(* Logix 5000 project; controller reports 1756-L63 rev 20.15; software revision 20.04; part 12 of 52 *)

        [360].log_data[14].valid := 1, [360].log_data[15].valid := 1, [360].log_data[16].valid := 1, [360].log_data[17].valid := 1, [360].log_data[18].valid := 1, [360].log_data[19].valid := 1, [360].time.Year := 2023, [360].time.Month := 1, [360].time.Day := 19, [360].time.Hour := 6, [360].time.Minute := 24, [360].time.Second := 59, [361].log_data[0].min := 1.0, [361].log_data[0].max := 1.0, [361].log_data[0].total := 300.0, [361].log_data[0].time := 300.0, [361].log_data[0].minminute := 25, [361].log_data[0].maxminute := 25, [361].log_data[0].valid := 1, [361].log_data[1].valid := 1, [361].log_data[2].valid := 1, [361].log_data[3].valid := 1, [361].log_data[4].valid := 1, [361].log_data[5].valid := 1, [361].log_data[6].valid := 1, [361].log_data[7].valid := 1, [361].log_data[8].valid := 1, [361].log_data[9].valid := 1, [361].log_data[10].valid := 1, [361].log_data[11].valid := 1, [361].log_data[12].valid := 1, [361].log_data[13].valid := 1, [361].log_data[14].valid := 1, [361].log_data[15].valid := 1, [361].log_data[16].valid := 1, [361].log_data[17].valid := 1, [361].log_data[18].valid := 1, [361].log_data[19].valid := 1, [361].time.Year := 2023, [361].time.Month := 1, [361].time.Day := 19, [361].time.Hour := 6, [361].time.Minute := 29, [361].time.Second := 59, [362].log_data[0].min := 1.0, [362].log_data[0].max := 1.0, [362].log_data[0].total := 300.0, [362].log_data[0].time := 300.0, [362].log_data[0].minminute := 30, [362].log_data[0].maxminute := 30, [362].log_data[0].valid := 1, [362].log_data[1].valid := 1, [362].log_data[2].valid := 1, [362].log_data[3].valid := 1, [362].log_data[4].valid := 1, [362].log_data[5].valid := 1, [362].log_data[6].valid := 1, [362].log_data[7].valid := 1, [362].log_data[8].valid := 1, [362].log_data[9].valid := 1,
        [362].log_data[10].valid := 1, [362].log_data[11].valid := 1, [362].log_data[12].valid := 1, [362].log_data[13].valid := 1, [362].log_data[14].valid := 1, [362].log_data[15].valid := 1, [362].log_data[16].valid := 1, [362].log_data[17].valid := 1, [362].log_data[18].valid := 1, [362].log_data[19].valid := 1, [362].time.Year := 2023, [362].time.Month := 1, [362].time.Day := 19, [362].time.Hour := 6, [362].time.Minute := 34, [362].time.Second := 59, [363].log_data[0].min := 1.0, [363].log_data[0].max := 1.0, [363].log_data[0].total := 300.0, [363].log_data[0].time := 300.0, [363].log_data[0].minminute := 35, [363].log_data[0].maxminute := 35, [363].log_data[0].valid := 1, [363].log_data[1].valid := 1, [363].log_data[2].valid := 1, [363].log_data[3].valid := 1, [363].log_data[4].valid := 1, [363].log_data[5].valid := 1, [363].log_data[6].valid := 1, [363].log_data[7].valid := 1, [363].log_data[8].valid := 1, [363].log_data[9].valid := 1, [363].log_data[10].valid := 1, [363].log_data[11].valid := 1, [363].log_data[12].valid := 1, [363].log_data[13].valid := 1, [363].log_data[14].valid := 1, [363].log_data[15].valid := 1, [363].log_data[16].valid := 1, [363].log_data[17].valid := 1, [363].log_data[18].valid := 1, [363].log_data[19].valid := 1, [363].time.Year := 2023, [363].time.Month := 1, [363].time.Day := 19, [363].time.Hour := 6, [363].time.Minute := 39, [363].time.Second := 59, [364].log_data[0].min := 1.0, [364].log_data[0].max := 1.0, [364].log_data[0].total := 300.0, [364].log_data[0].time := 300.0, [364].log_data[0].minminute := 40, [364].log_data[0].maxminute := 40, [364].log_data[0].valid := 1, [364].log_data[1].valid := 1, [364].log_data[2].valid := 1, [364].log_data[3].valid := 1, [364].log_data[4].valid := 1, [364].log_data[5].valid := 1,
        [364].log_data[6].valid := 1, [364].log_data[7].valid := 1, [364].log_data[8].valid := 1, [364].log_data[9].valid := 1, [364].log_data[10].valid := 1, [364].log_data[11].valid := 1, [364].log_data[12].valid := 1, [364].log_data[13].valid := 1, [364].log_data[14].valid := 1, [364].log_data[15].valid := 1, [364].log_data[16].valid := 1, [364].log_data[17].valid := 1, [364].log_data[18].valid := 1, [364].log_data[19].valid := 1, [364].time.Year := 2023, [364].time.Month := 1, [364].time.Day := 19, [364].time.Hour := 6, [364].time.Minute := 44, [364].time.Second := 59, [365].log_data[0].min := 1.0, [365].log_data[0].max := 1.0, [365].log_data[0].total := 300.0, [365].log_data[0].time := 300.0, [365].log_data[0].minminute := 45, [365].log_data[0].maxminute := 45, [365].log_data[0].valid := 1, [365].log_data[1].valid := 1, [365].log_data[2].valid := 1, [365].log_data[3].valid := 1, [365].log_data[4].valid := 1, [365].log_data[5].valid := 1, [365].log_data[6].valid := 1, [365].log_data[7].valid := 1, [365].log_data[8].valid := 1, [365].log_data[9].valid := 1, [365].log_data[10].valid := 1, [365].log_data[11].valid := 1, [365].log_data[12].valid := 1, [365].log_data[13].valid := 1, [365].log_data[14].valid := 1, [365].log_data[15].valid := 1, [365].log_data[16].valid := 1, [365].log_data[17].valid := 1, [365].log_data[18].valid := 1, [365].log_data[19].valid := 1, [365].time.Year := 2023, [365].time.Month := 1, [365].time.Day := 19, [365].time.Hour := 6, [365].time.Minute := 49, [365].time.Second := 59, [366].log_data[0].min := 1.0, [366].log_data[0].max := 1.0, [366].log_data[0].total := 300.0, [366].log_data[0].time := 300.0, [366].log_data[0].minminute := 50, [366].log_data[0].maxminute := 50, [366].log_data[0].valid := 1, [366].log_data[1].valid := 1,
        [366].log_data[2].valid := 1, [366].log_data[3].valid := 1, [366].log_data[4].valid := 1, [366].log_data[5].valid := 1, [366].log_data[6].valid := 1, [366].log_data[7].valid := 1, [366].log_data[8].valid := 1, [366].log_data[9].valid := 1, [366].log_data[10].valid := 1, [366].log_data[11].valid := 1, [366].log_data[12].valid := 1, [366].log_data[13].valid := 1, [366].log_data[14].valid := 1, [366].log_data[15].valid := 1, [366].log_data[16].valid := 1, [366].log_data[17].valid := 1, [366].log_data[18].valid := 1, [366].log_data[19].valid := 1, [366].time.Year := 2023, [366].time.Month := 1, [366].time.Day := 19, [366].time.Hour := 6, [366].time.Minute := 54, [366].time.Second := 59, [367].log_data[0].min := 1.0, [367].log_data[0].max := 1.0, [367].log_data[0].total := 300.0, [367].log_data[0].time := 300.0, [367].log_data[0].minminute := 55, [367].log_data[0].maxminute := 55, [367].log_data[0].valid := 1, [367].log_data[1].valid := 1, [367].log_data[2].valid := 1, [367].log_data[3].valid := 1, [367].log_data[4].valid := 1, [367].log_data[5].valid := 1, [367].log_data[6].valid := 1, [367].log_data[7].valid := 1, [367].log_data[8].valid := 1, [367].log_data[9].valid := 1, [367].log_data[10].valid := 1, [367].log_data[11].valid := 1, [367].log_data[12].valid := 1, [367].log_data[13].valid := 1, [367].log_data[14].valid := 1, [367].log_data[15].valid := 1, [367].log_data[16].valid := 1, [367].log_data[17].valid := 1, [367].log_data[18].valid := 1, [367].log_data[19].valid := 1, [367].time.Year := 2023, [367].time.Month := 1, [367].time.Day := 19, [367].time.Hour := 6, [367].time.Minute := 59, [367].time.Second := 59, [368].log_data[0].min := 1.0, [368].log_data[0].max := 1.0, [368].log_data[0].total := 300.0, [368].log_data[0].time := 300.0,
        [368].log_data[0].valid := 1, [368].log_data[1].valid := 1, [368].log_data[2].valid := 1, [368].log_data[3].valid := 1, [368].log_data[4].valid := 1, [368].log_data[5].valid := 1, [368].log_data[6].valid := 1, [368].log_data[7].valid := 1, [368].log_data[8].valid := 1, [368].log_data[9].valid := 1, [368].log_data[10].valid := 1, [368].log_data[11].valid := 1, [368].log_data[12].valid := 1, [368].log_data[13].valid := 1, [368].log_data[14].valid := 1, [368].log_data[15].valid := 1, [368].log_data[16].valid := 1, [368].log_data[17].valid := 1, [368].log_data[18].valid := 1, [368].log_data[19].valid := 1, [368].time.Year := 2023, [368].time.Month := 1, [368].time.Day := 19, [368].time.Hour := 7, [368].time.Minute := 4, [368].time.Second := 59, [369].log_data[0].min := 1.0, [369].log_data[0].max := 1.0, [369].log_data[0].total := 300.0, [369].log_data[0].time := 300.0, [369].log_data[0].minminute := 5, [369].log_data[0].maxminute := 5, [369].log_data[0].valid := 1, [369].log_data[1].valid := 1, [369].log_data[2].valid := 1, [369].log_data[3].valid := 1, [369].log_data[4].valid := 1, [369].log_data[5].valid := 1, [369].log_data[6].valid := 1, [369].log_data[7].valid := 1, [369].log_data[8].valid := 1, [369].log_data[9].valid := 1, [369].log_data[10].valid := 1, [369].log_data[11].valid := 1, [369].log_data[12].valid := 1, [369].log_data[13].valid := 1, [369].log_data[14].valid := 1, [369].log_data[15].valid := 1, [369].log_data[16].valid := 1, [369].log_data[17].valid := 1, [369].log_data[18].valid := 1, [369].log_data[19].valid := 1, [369].time.Year := 2023, [369].time.Month := 1, [369].time.Day := 19, [369].time.Hour := 7, [369].time.Minute := 9, [369].time.Second := 59, [370].log_data[0].min := 1.0, [370].log_data[0].max := 1.0,
        [370].log_data[0].total := 300.0, [370].log_data[0].time := 300.0, [370].log_data[0].minminute := 10, [370].log_data[0].maxminute := 10, [370].log_data[0].valid := 1, [370].log_data[1].valid := 1, [370].log_data[2].valid := 1, [370].log_data[3].valid := 1, [370].log_data[4].valid := 1, [370].log_data[5].valid := 1, [370].log_data[6].valid := 1, [370].log_data[7].valid := 1, [370].log_data[8].valid := 1, [370].log_data[9].valid := 1, [370].log_data[10].valid := 1, [370].log_data[11].valid := 1, [370].log_data[12].valid := 1, [370].log_data[13].valid := 1, [370].log_data[14].valid := 1, [370].log_data[15].valid := 1, [370].log_data[16].valid := 1, [370].log_data[17].valid := 1, [370].log_data[18].valid := 1, [370].log_data[19].valid := 1, [370].time.Year := 2023, [370].time.Month := 1, [370].time.Day := 19, [370].time.Hour := 7, [370].time.Minute := 14, [370].time.Second := 59, [371].log_data[0].min := 1.0, [371].log_data[0].max := 1.0, [371].log_data[0].total := 300.0, [371].log_data[0].time := 300.0, [371].log_data[0].minminute := 15, [371].log_data[0].maxminute := 15, [371].log_data[0].valid := 1, [371].log_data[1].valid := 1, [371].log_data[2].valid := 1, [371].log_data[3].valid := 1, [371].log_data[4].valid := 1, [371].log_data[5].valid := 1, [371].log_data[6].valid := 1, [371].log_data[7].valid := 1, [371].log_data[8].valid := 1, [371].log_data[9].valid := 1, [371].log_data[10].valid := 1, [371].log_data[11].valid := 1, [371].log_data[12].valid := 1, [371].log_data[13].valid := 1, [371].log_data[14].valid := 1, [371].log_data[15].valid := 1, [371].log_data[16].valid := 1, [371].log_data[17].valid := 1, [371].log_data[18].valid := 1, [371].log_data[19].valid := 1, [371].time.Year := 2023, [371].time.Month := 1, [371].time.Day := 19, [371].time.Hour := 7,
        [371].time.Minute := 19, [371].time.Second := 59, [372].log_data[0].min := 1.0, [372].log_data[0].max := 1.0, [372].log_data[0].total := 300.0, [372].log_data[0].time := 300.0, [372].log_data[0].minminute := 20, [372].log_data[0].maxminute := 20, [372].log_data[0].valid := 1, [372].log_data[1].valid := 1, [372].log_data[2].valid := 1, [372].log_data[3].valid := 1, [372].log_data[4].valid := 1, [372].log_data[5].valid := 1, [372].log_data[6].valid := 1, [372].log_data[7].valid := 1, [372].log_data[8].valid := 1, [372].log_data[9].valid := 1, [372].log_data[10].valid := 1, [372].log_data[11].valid := 1, [372].log_data[12].valid := 1, [372].log_data[13].valid := 1, [372].log_data[14].valid := 1, [372].log_data[15].valid := 1, [372].log_data[16].valid := 1, [372].log_data[17].valid := 1, [372].log_data[18].valid := 1, [372].log_data[19].valid := 1, [372].time.Year := 2023, [372].time.Month := 1, [372].time.Day := 19, [372].time.Hour := 7, [372].time.Minute := 24, [372].time.Second := 59, [373].log_data[0].min := 1.0, [373].log_data[0].max := 1.0, [373].log_data[0].total := 300.0, [373].log_data[0].time := 300.0, [373].log_data[0].minminute := 25, [373].log_data[0].maxminute := 25, [373].log_data[0].valid := 1, [373].log_data[1].valid := 1, [373].log_data[2].valid := 1, [373].log_data[3].valid := 1, [373].log_data[4].valid := 1, [373].log_data[5].valid := 1, [373].log_data[6].valid := 1, [373].log_data[7].valid := 1, [373].log_data[8].valid := 1, [373].log_data[9].valid := 1, [373].log_data[10].valid := 1, [373].log_data[11].valid := 1, [373].log_data[12].valid := 1, [373].log_data[13].valid := 1, [373].log_data[14].valid := 1, [373].log_data[15].valid := 1, [373].log_data[16].valid := 1, [373].log_data[17].valid := 1, [373].log_data[18].valid := 1, [373].log_data[19].valid := 1,
        [373].time.Year := 2023, [373].time.Month := 1, [373].time.Day := 19, [373].time.Hour := 7, [373].time.Minute := 29, [373].time.Second := 59, [374].log_data[0].min := 1.0, [374].log_data[0].max := 1.0, [374].log_data[0].total := 300.0, [374].log_data[0].time := 300.0, [374].log_data[0].minminute := 30, [374].log_data[0].maxminute := 30, [374].log_data[0].valid := 1, [374].log_data[1].valid := 1, [374].log_data[2].valid := 1, [374].log_data[3].valid := 1, [374].log_data[4].valid := 1, [374].log_data[5].valid := 1, [374].log_data[6].valid := 1, [374].log_data[7].valid := 1, [374].log_data[8].valid := 1, [374].log_data[9].valid := 1, [374].log_data[10].valid := 1, [374].log_data[11].valid := 1, [374].log_data[12].valid := 1, [374].log_data[13].valid := 1, [374].log_data[14].valid := 1, [374].log_data[15].valid := 1, [374].log_data[16].valid := 1, [374].log_data[17].valid := 1, [374].log_data[18].valid := 1, [374].log_data[19].valid := 1, [374].time.Year := 2023, [374].time.Month := 1, [374].time.Day := 19, [374].time.Hour := 7, [374].time.Minute := 34, [374].time.Second := 59, [375].log_data[0].min := 1.0, [375].log_data[0].max := 1.0, [375].log_data[0].total := 300.0, [375].log_data[0].time := 300.0, [375].log_data[0].minminute := 35, [375].log_data[0].maxminute := 35, [375].log_data[0].valid := 1, [375].log_data[1].valid := 1, [375].log_data[2].valid := 1, [375].log_data[3].valid := 1, [375].log_data[4].valid := 1, [375].log_data[5].valid := 1, [375].log_data[6].valid := 1, [375].log_data[7].valid := 1, [375].log_data[8].valid := 1, [375].log_data[9].valid := 1, [375].log_data[10].valid := 1, [375].log_data[11].valid := 1, [375].log_data[12].valid := 1, [375].log_data[13].valid := 1, [375].log_data[14].valid := 1, [375].log_data[15].valid := 1,
        [375].log_data[16].valid := 1, [375].log_data[17].valid := 1, [375].log_data[18].valid := 1, [375].log_data[19].valid := 1, [375].time.Year := 2023, [375].time.Month := 1, [375].time.Day := 19, [375].time.Hour := 7, [375].time.Minute := 39, [375].time.Second := 59, [376].log_data[0].min := 1.0, [376].log_data[0].max := 1.0, [376].log_data[0].total := 300.0, [376].log_data[0].time := 300.0, [376].log_data[0].minminute := 40, [376].log_data[0].maxminute := 40, [376].log_data[0].valid := 1, [376].log_data[1].valid := 1, [376].log_data[2].valid := 1, [376].log_data[3].valid := 1, [376].log_data[4].valid := 1, [376].log_data[5].valid := 1, [376].log_data[6].valid := 1, [376].log_data[7].valid := 1, [376].log_data[8].valid := 1, [376].log_data[9].valid := 1, [376].log_data[10].valid := 1, [376].log_data[11].valid := 1, [376].log_data[12].valid := 1, [376].log_data[13].valid := 1, [376].log_data[14].valid := 1, [376].log_data[15].valid := 1, [376].log_data[16].valid := 1, [376].log_data[17].valid := 1, [376].log_data[18].valid := 1, [376].log_data[19].valid := 1, [376].time.Year := 2023, [376].time.Month := 1, [376].time.Day := 19, [376].time.Hour := 7, [376].time.Minute := 44, [376].time.Second := 59, [377].log_data[0].min := 1.0, [377].log_data[0].max := 1.0, [377].log_data[0].total := 300.0, [377].log_data[0].time := 300.0, [377].log_data[0].minminute := 45, [377].log_data[0].maxminute := 45, [377].log_data[0].valid := 1, [377].log_data[1].valid := 1, [377].log_data[2].valid := 1, [377].log_data[3].valid := 1, [377].log_data[4].valid := 1, [377].log_data[5].valid := 1, [377].log_data[6].valid := 1, [377].log_data[7].valid := 1, [377].log_data[8].valid := 1, [377].log_data[9].valid := 1, [377].log_data[10].valid := 1, [377].log_data[11].valid := 1,
        [377].log_data[12].valid := 1, [377].log_data[13].valid := 1, [377].log_data[14].valid := 1, [377].log_data[15].valid := 1, [377].log_data[16].valid := 1, [377].log_data[17].valid := 1, [377].log_data[18].valid := 1, [377].log_data[19].valid := 1, [377].time.Year := 2023, [377].time.Month := 1, [377].time.Day := 19, [377].time.Hour := 7, [377].time.Minute := 49, [377].time.Second := 59, [378].log_data[0].min := 1.0, [378].log_data[0].max := 1.0, [378].log_data[0].total := 300.0, [378].log_data[0].time := 300.0, [378].log_data[0].minminute := 50, [378].log_data[0].maxminute := 50, [378].log_data[0].valid := 1, [378].log_data[1].valid := 1, [378].log_data[2].valid := 1, [378].log_data[3].valid := 1, [378].log_data[4].valid := 1, [378].log_data[5].valid := 1, [378].log_data[6].valid := 1, [378].log_data[7].valid := 1, [378].log_data[8].valid := 1, [378].log_data[9].valid := 1, [378].log_data[10].valid := 1, [378].log_data[11].valid := 1, [378].log_data[12].valid := 1, [378].log_data[13].valid := 1, [378].log_data[14].valid := 1, [378].log_data[15].valid := 1, [378].log_data[16].valid := 1, [378].log_data[17].valid := 1, [378].log_data[18].valid := 1, [378].log_data[19].valid := 1, [378].time.Year := 2023, [378].time.Month := 1, [378].time.Day := 19, [378].time.Hour := 7, [378].time.Minute := 54, [378].time.Second := 59, [379].log_data[0].min := 1.0, [379].log_data[0].max := 1.0, [379].log_data[0].total := 300.0, [379].log_data[0].time := 300.0, [379].log_data[0].minminute := 55, [379].log_data[0].maxminute := 55, [379].log_data[0].valid := 1, [379].log_data[1].valid := 1, [379].log_data[2].valid := 1, [379].log_data[3].valid := 1, [379].log_data[4].valid := 1, [379].log_data[5].valid := 1, [379].log_data[6].valid := 1, [379].log_data[7].valid := 1,
        [379].log_data[8].valid := 1, [379].log_data[9].valid := 1, [379].log_data[10].valid := 1, [379].log_data[11].valid := 1, [379].log_data[12].valid := 1, [379].log_data[13].valid := 1, [379].log_data[14].valid := 1, [379].log_data[15].valid := 1, [379].log_data[16].valid := 1, [379].log_data[17].valid := 1, [379].log_data[18].valid := 1, [379].log_data[19].valid := 1, [379].time.Year := 2023, [379].time.Month := 1, [379].time.Day := 19, [379].time.Hour := 7, [379].time.Minute := 59, [379].time.Second := 59, [380].log_data[0].min := 1.0, [380].log_data[0].max := 1.0, [380].log_data[0].total := 299.5, [380].log_data[0].time := 299.5, [380].log_data[0].valid := 1, [380].log_data[1].valid := 1, [380].log_data[2].valid := 1, [380].log_data[3].valid := 1, [380].log_data[4].valid := 1, [380].log_data[5].valid := 1, [380].log_data[6].valid := 1, [380].log_data[7].valid := 1, [380].log_data[8].valid := 1, [380].log_data[9].valid := 1, [380].log_data[10].valid := 1, [380].log_data[11].valid := 1, [380].log_data[12].valid := 1, [380].log_data[13].valid := 1, [380].log_data[14].valid := 1, [380].log_data[15].valid := 1, [380].log_data[16].valid := 1, [380].log_data[17].valid := 1, [380].log_data[18].valid := 1, [380].log_data[19].valid := 1, [380].time.Year := 2023, [380].time.Month := 1, [380].time.Day := 19, [380].time.Hour := 8, [380].time.Minute := 4, [380].time.Second := 59, [381].log_data[0].min := 1.0, [381].log_data[0].max := 1.0, [381].log_data[0].total := 300.0, [381].log_data[0].time := 300.0, [381].log_data[0].minminute := 5, [381].log_data[0].maxminute := 5, [381].log_data[0].valid := 1, [381].log_data[1].valid := 1, [381].log_data[2].valid := 1, [381].log_data[3].valid := 1, [381].log_data[4].valid := 1, [381].log_data[5].valid := 1,
        [381].log_data[6].valid := 1, [381].log_data[7].valid := 1, [381].log_data[8].valid := 1, [381].log_data[9].valid := 1, [381].log_data[10].valid := 1, [381].log_data[11].valid := 1, [381].log_data[12].valid := 1, [381].log_data[13].valid := 1, [381].log_data[14].valid := 1, [381].log_data[15].valid := 1, [381].log_data[16].valid := 1, [381].log_data[17].valid := 1, [381].log_data[18].valid := 1, [381].log_data[19].valid := 1, [381].time.Year := 2023, [381].time.Month := 1, [381].time.Day := 19, [381].time.Hour := 8, [381].time.Minute := 9, [381].time.Second := 59, [382].log_data[0].min := 1.0, [382].log_data[0].max := 1.0, [382].log_data[0].total := 300.0, [382].log_data[0].time := 300.0, [382].log_data[0].minminute := 10, [382].log_data[0].maxminute := 10, [382].log_data[0].valid := 1, [382].log_data[1].valid := 1, [382].log_data[2].valid := 1, [382].log_data[3].valid := 1, [382].log_data[4].valid := 1, [382].log_data[5].valid := 1, [382].log_data[6].valid := 1, [382].log_data[7].valid := 1, [382].log_data[8].valid := 1, [382].log_data[9].valid := 1, [382].log_data[10].valid := 1, [382].log_data[11].valid := 1, [382].log_data[12].valid := 1, [382].log_data[13].valid := 1, [382].log_data[14].valid := 1, [382].log_data[15].valid := 1, [382].log_data[16].valid := 1, [382].log_data[17].valid := 1, [382].log_data[18].valid := 1, [382].log_data[19].valid := 1, [382].time.Year := 2023, [382].time.Month := 1, [382].time.Day := 19, [382].time.Hour := 8, [382].time.Minute := 14, [382].time.Second := 59, [383].log_data[0].min := 1.0, [383].log_data[0].max := 1.0, [383].log_data[0].total := 300.0, [383].log_data[0].time := 300.0, [383].log_data[0].minminute := 15, [383].log_data[0].maxminute := 15, [383].log_data[0].valid := 1, [383].log_data[1].valid := 1,
        [383].log_data[2].valid := 1, [383].log_data[3].valid := 1, [383].log_data[4].valid := 1, [383].log_data[5].valid := 1, [383].log_data[6].valid := 1, [383].log_data[7].valid := 1, [383].log_data[8].valid := 1, [383].log_data[9].valid := 1, [383].log_data[10].valid := 1, [383].log_data[11].valid := 1, [383].log_data[12].valid := 1, [383].log_data[13].valid := 1, [383].log_data[14].valid := 1, [383].log_data[15].valid := 1, [383].log_data[16].valid := 1, [383].log_data[17].valid := 1, [383].log_data[18].valid := 1, [383].log_data[19].valid := 1, [383].time.Year := 2023, [383].time.Month := 1, [383].time.Day := 19, [383].time.Hour := 8, [383].time.Minute := 19, [383].time.Second := 59, [384].log_data[0].min := 1.0, [384].log_data[0].max := 1.0, [384].log_data[0].total := 300.0, [384].log_data[0].time := 300.0, [384].log_data[0].minminute := 20, [384].log_data[0].maxminute := 20, [384].log_data[0].valid := 1, [384].log_data[1].valid := 1, [384].log_data[2].valid := 1, [384].log_data[3].valid := 1, [384].log_data[4].valid := 1, [384].log_data[5].valid := 1, [384].log_data[6].valid := 1, [384].log_data[7].valid := 1, [384].log_data[8].valid := 1, [384].log_data[9].valid := 1, [384].log_data[10].valid := 1, [384].log_data[11].valid := 1, [384].log_data[12].valid := 1, [384].log_data[13].valid := 1, [384].log_data[14].valid := 1, [384].log_data[15].valid := 1, [384].log_data[16].valid := 1, [384].log_data[17].valid := 1, [384].log_data[18].valid := 1, [384].log_data[19].valid := 1, [384].time.Year := 2023, [384].time.Month := 1, [384].time.Day := 19, [384].time.Hour := 8, [384].time.Minute := 24, [384].time.Second := 59, [385].log_data[0].min := 1.0, [385].log_data[0].max := 1.0, [385].log_data[0].total := 300.0, [385].log_data[0].time := 300.0,
        [385].log_data[0].minminute := 25, [385].log_data[0].maxminute := 25, [385].log_data[0].valid := 1, [385].log_data[1].valid := 1, [385].log_data[2].valid := 1, [385].log_data[3].valid := 1, [385].log_data[4].valid := 1, [385].log_data[5].valid := 1, [385].log_data[6].valid := 1, [385].log_data[7].valid := 1, [385].log_data[8].valid := 1, [385].log_data[9].valid := 1, [385].log_data[10].valid := 1, [385].log_data[11].valid := 1, [385].log_data[12].valid := 1, [385].log_data[13].valid := 1, [385].log_data[14].valid := 1, [385].log_data[15].valid := 1, [385].log_data[16].valid := 1, [385].log_data[17].valid := 1, [385].log_data[18].valid := 1, [385].log_data[19].valid := 1, [385].time.Year := 2023, [385].time.Month := 1, [385].time.Day := 19, [385].time.Hour := 8, [385].time.Minute := 29, [385].time.Second := 59, [386].log_data[0].min := 1.0, [386].log_data[0].max := 1.0, [386].log_data[0].total := 300.0, [386].log_data[0].time := 300.0, [386].log_data[0].minminute := 30, [386].log_data[0].maxminute := 30, [386].log_data[0].valid := 1, [386].log_data[1].valid := 1, [386].log_data[2].valid := 1, [386].log_data[3].valid := 1, [386].log_data[4].valid := 1, [386].log_data[5].valid := 1, [386].log_data[6].valid := 1, [386].log_data[7].valid := 1, [386].log_data[8].valid := 1, [386].log_data[9].valid := 1, [386].log_data[10].valid := 1, [386].log_data[11].valid := 1, [386].log_data[12].valid := 1, [386].log_data[13].valid := 1, [386].log_data[14].valid := 1, [386].log_data[15].valid := 1, [386].log_data[16].valid := 1, [386].log_data[17].valid := 1, [386].log_data[18].valid := 1, [386].log_data[19].valid := 1, [386].time.Year := 2023, [386].time.Month := 1, [386].time.Day := 19, [386].time.Hour := 8, [386].time.Minute := 34, [386].time.Second := 59,
        [387].log_data[0].min := 1.0, [387].log_data[0].max := 1.0, [387].log_data[0].total := 300.0, [387].log_data[0].time := 300.0, [387].log_data[0].minminute := 35, [387].log_data[0].maxminute := 35, [387].log_data[0].valid := 1, [387].log_data[1].valid := 1, [387].log_data[2].valid := 1, [387].log_data[3].valid := 1, [387].log_data[4].valid := 1, [387].log_data[5].valid := 1, [387].log_data[6].valid := 1, [387].log_data[7].valid := 1, [387].log_data[8].valid := 1, [387].log_data[9].valid := 1, [387].log_data[10].valid := 1, [387].log_data[11].valid := 1, [387].log_data[12].valid := 1, [387].log_data[13].valid := 1, [387].log_data[14].valid := 1, [387].log_data[15].valid := 1, [387].log_data[16].valid := 1, [387].log_data[17].valid := 1, [387].log_data[18].valid := 1, [387].log_data[19].valid := 1, [387].time.Year := 2023, [387].time.Month := 1, [387].time.Day := 19, [387].time.Hour := 8, [387].time.Minute := 39, [387].time.Second := 59, [388].log_data[0].min := 1.0, [388].log_data[0].max := 1.0, [388].log_data[0].total := 300.0, [388].log_data[0].time := 300.0, [388].log_data[0].minminute := 40, [388].log_data[0].maxminute := 40, [388].log_data[0].valid := 1, [388].log_data[1].valid := 1, [388].log_data[2].valid := 1, [388].log_data[3].valid := 1, [388].log_data[4].valid := 1, [388].log_data[5].valid := 1, [388].log_data[6].valid := 1, [388].log_data[7].valid := 1, [388].log_data[8].valid := 1, [388].log_data[9].valid := 1, [388].log_data[10].valid := 1, [388].log_data[11].valid := 1, [388].log_data[12].valid := 1, [388].log_data[13].valid := 1, [388].log_data[14].valid := 1, [388].log_data[15].valid := 1, [388].log_data[16].valid := 1, [388].log_data[17].valid := 1, [388].log_data[18].valid := 1, [388].log_data[19].valid := 1, [388].time.Year := 2023, [388].time.Month := 1,
        [388].time.Day := 19, [388].time.Hour := 8, [388].time.Minute := 44, [388].time.Second := 59, [389].log_data[0].min := 1.0, [389].log_data[0].max := 1.0, [389].log_data[0].total := 300.0, [389].log_data[0].time := 300.0, [389].log_data[0].minminute := 45, [389].log_data[0].maxminute := 45, [389].log_data[0].valid := 1, [389].log_data[1].valid := 1, [389].log_data[2].valid := 1, [389].log_data[3].valid := 1, [389].log_data[4].valid := 1, [389].log_data[5].valid := 1, [389].log_data[6].valid := 1, [389].log_data[7].valid := 1, [389].log_data[8].valid := 1, [389].log_data[9].valid := 1, [389].log_data[10].valid := 1, [389].log_data[11].valid := 1, [389].log_data[12].valid := 1, [389].log_data[13].valid := 1, [389].log_data[14].valid := 1, [389].log_data[15].valid := 1, [389].log_data[16].valid := 1, [389].log_data[17].valid := 1, [389].log_data[18].valid := 1, [389].log_data[19].valid := 1, [389].time.Year := 2023, [389].time.Month := 1, [389].time.Day := 19, [389].time.Hour := 8, [389].time.Minute := 49, [389].time.Second := 59, [390].log_data[0].min := 1.0, [390].log_data[0].max := 1.0, [390].log_data[0].total := 300.0, [390].log_data[0].time := 300.0, [390].log_data[0].minminute := 50, [390].log_data[0].maxminute := 50, [390].log_data[0].valid := 1, [390].log_data[1].valid := 1, [390].log_data[2].valid := 1, [390].log_data[3].valid := 1, [390].log_data[4].valid := 1, [390].log_data[5].valid := 1, [390].log_data[6].valid := 1, [390].log_data[7].valid := 1, [390].log_data[8].valid := 1, [390].log_data[9].valid := 1, [390].log_data[10].valid := 1, [390].log_data[11].valid := 1, [390].log_data[12].valid := 1, [390].log_data[13].valid := 1, [390].log_data[14].valid := 1, [390].log_data[15].valid := 1, [390].log_data[16].valid := 1, [390].log_data[17].valid := 1,
        [390].log_data[18].valid := 1, [390].log_data[19].valid := 1, [390].time.Year := 2023, [390].time.Month := 1, [390].time.Day := 19, [390].time.Hour := 8, [390].time.Minute := 54, [390].time.Second := 59, [391].log_data[0].min := 1.0, [391].log_data[0].max := 1.0, [391].log_data[0].total := 300.0, [391].log_data[0].time := 300.0, [391].log_data[0].minminute := 55, [391].log_data[0].maxminute := 55, [391].log_data[0].valid := 1, [391].log_data[1].valid := 1, [391].log_data[2].valid := 1, [391].log_data[3].valid := 1, [391].log_data[4].valid := 1, [391].log_data[5].valid := 1, [391].log_data[6].valid := 1, [391].log_data[7].valid := 1, [391].log_data[8].valid := 1, [391].log_data[9].valid := 1, [391].log_data[10].valid := 1, [391].log_data[11].valid := 1, [391].log_data[12].valid := 1, [391].log_data[13].valid := 1, [391].log_data[14].valid := 1, [391].log_data[15].valid := 1, [391].log_data[16].valid := 1, [391].log_data[17].valid := 1, [391].log_data[18].valid := 1, [391].log_data[19].valid := 1, [391].time.Year := 2023, [391].time.Month := 1, [391].time.Day := 19, [391].time.Hour := 8, [391].time.Minute := 59, [391].time.Second := 59, [392].log_data[0].min := 1.0, [392].log_data[0].max := 1.0, [392].log_data[0].total := 300.0, [392].log_data[0].time := 300.0, [392].log_data[0].valid := 1, [392].log_data[1].valid := 1, [392].log_data[2].valid := 1, [392].log_data[3].valid := 1, [392].log_data[4].valid := 1, [392].log_data[5].valid := 1, [392].log_data[6].valid := 1, [392].log_data[7].valid := 1, [392].log_data[8].valid := 1, [392].log_data[9].valid := 1, [392].log_data[10].valid := 1, [392].log_data[11].valid := 1, [392].log_data[12].valid := 1, [392].log_data[13].valid := 1, [392].log_data[14].valid := 1, [392].log_data[15].valid := 1,
        [392].log_data[16].valid := 1, [392].log_data[17].valid := 1, [392].log_data[18].valid := 1, [392].log_data[19].valid := 1, [392].time.Year := 2023, [392].time.Month := 1, [392].time.Day := 19, [392].time.Hour := 9, [392].time.Minute := 4, [392].time.Second := 59, [393].log_data[0].min := 1.0, [393].log_data[0].max := 1.0, [393].log_data[0].total := 300.0, [393].log_data[0].time := 300.0, [393].log_data[0].minminute := 5, [393].log_data[0].maxminute := 5, [393].log_data[0].valid := 1, [393].log_data[1].valid := 1, [393].log_data[2].valid := 1, [393].log_data[3].valid := 1, [393].log_data[4].valid := 1, [393].log_data[5].valid := 1, [393].log_data[6].valid := 1, [393].log_data[7].valid := 1, [393].log_data[8].valid := 1, [393].log_data[9].valid := 1, [393].log_data[10].valid := 1, [393].log_data[11].valid := 1, [393].log_data[12].valid := 1, [393].log_data[13].valid := 1, [393].log_data[14].valid := 1, [393].log_data[15].valid := 1, [393].log_data[16].valid := 1, [393].log_data[17].valid := 1, [393].log_data[18].valid := 1, [393].log_data[19].valid := 1, [393].time.Year := 2023, [393].time.Month := 1, [393].time.Day := 19, [393].time.Hour := 9, [393].time.Minute := 9, [393].time.Second := 59, [394].log_data[0].min := 1.0, [394].log_data[0].max := 1.0, [394].log_data[0].total := 300.0, [394].log_data[0].time := 300.0, [394].log_data[0].minminute := 10, [394].log_data[0].maxminute := 10, [394].log_data[0].valid := 1, [394].log_data[1].valid := 1, [394].log_data[2].valid := 1, [394].log_data[3].valid := 1, [394].log_data[4].valid := 1, [394].log_data[5].valid := 1, [394].log_data[6].valid := 1, [394].log_data[7].valid := 1, [394].log_data[8].valid := 1, [394].log_data[9].valid := 1, [394].log_data[10].valid := 1, [394].log_data[11].valid := 1,
        [394].log_data[12].valid := 1, [394].log_data[13].valid := 1, [394].log_data[14].valid := 1, [394].log_data[15].valid := 1, [394].log_data[16].valid := 1, [394].log_data[17].valid := 1, [394].log_data[18].valid := 1, [394].log_data[19].valid := 1, [394].time.Year := 2023, [394].time.Month := 1, [394].time.Day := 19, [394].time.Hour := 9, [394].time.Minute := 14, [394].time.Second := 59, [395].log_data[0].min := 1.0, [395].log_data[0].max := 1.0, [395].log_data[0].total := 300.0, [395].log_data[0].time := 300.0, [395].log_data[0].minminute := 15, [395].log_data[0].maxminute := 15, [395].log_data[0].valid := 1, [395].log_data[1].valid := 1, [395].log_data[2].valid := 1, [395].log_data[3].valid := 1, [395].log_data[4].valid := 1, [395].log_data[5].valid := 1, [395].log_data[6].valid := 1, [395].log_data[7].valid := 1, [395].log_data[8].valid := 1, [395].log_data[9].valid := 1, [395].log_data[10].valid := 1, [395].log_data[11].valid := 1, [395].log_data[12].valid := 1, [395].log_data[13].valid := 1, [395].log_data[14].valid := 1, [395].log_data[15].valid := 1, [395].log_data[16].valid := 1, [395].log_data[17].valid := 1, [395].log_data[18].valid := 1, [395].log_data[19].valid := 1, [395].time.Year := 2023, [395].time.Month := 1, [395].time.Day := 19, [395].time.Hour := 9, [395].time.Minute := 19, [395].time.Second := 59, [396].log_data[0].min := 1.0, [396].log_data[0].max := 1.0, [396].log_data[0].total := 300.0, [396].log_data[0].time := 300.0, [396].log_data[0].minminute := 20, [396].log_data[0].maxminute := 20, [396].log_data[0].valid := 1, [396].log_data[1].valid := 1, [396].log_data[2].valid := 1, [396].log_data[3].valid := 1, [396].log_data[4].valid := 1, [396].log_data[5].valid := 1, [396].log_data[6].valid := 1, [396].log_data[7].valid := 1,
        [396].log_data[8].valid := 1, [396].log_data[9].valid := 1, [396].log_data[10].valid := 1, [396].log_data[11].valid := 1, [396].log_data[12].valid := 1, [396].log_data[13].valid := 1, [396].log_data[14].valid := 1, [396].log_data[15].valid := 1, [396].log_data[16].valid := 1, [396].log_data[17].valid := 1, [396].log_data[18].valid := 1, [396].log_data[19].valid := 1, [396].time.Year := 2023, [396].time.Month := 1, [396].time.Day := 19, [396].time.Hour := 9, [396].time.Minute := 24, [396].time.Second := 59, [397].log_data[0].min := 1.0, [397].log_data[0].max := 1.0, [397].log_data[0].total := 300.0, [397].log_data[0].time := 300.0, [397].log_data[0].minminute := 25, [397].log_data[0].maxminute := 25, [397].log_data[0].valid := 1, [397].log_data[1].valid := 1, [397].log_data[2].valid := 1, [397].log_data[3].valid := 1, [397].log_data[4].valid := 1, [397].log_data[5].valid := 1, [397].log_data[6].valid := 1, [397].log_data[7].valid := 1, [397].log_data[8].valid := 1, [397].log_data[9].valid := 1, [397].log_data[10].valid := 1, [397].log_data[11].valid := 1, [397].log_data[12].valid := 1, [397].log_data[13].valid := 1, [397].log_data[14].valid := 1, [397].log_data[15].valid := 1, [397].log_data[16].valid := 1, [397].log_data[17].valid := 1, [397].log_data[18].valid := 1, [397].log_data[19].valid := 1, [397].time.Year := 2023, [397].time.Month := 1, [397].time.Day := 19, [397].time.Hour := 9, [397].time.Minute := 29, [397].time.Second := 59, [398].log_data[0].min := 1.0, [398].log_data[0].max := 1.0, [398].log_data[0].total := 300.0, [398].log_data[0].time := 300.0, [398].log_data[0].minminute := 30, [398].log_data[0].maxminute := 30, [398].log_data[0].valid := 1, [398].log_data[1].valid := 1, [398].log_data[2].valid := 1, [398].log_data[3].valid := 1,
        [398].log_data[4].valid := 1, [398].log_data[5].valid := 1, [398].log_data[6].valid := 1, [398].log_data[7].valid := 1, [398].log_data[8].valid := 1, [398].log_data[9].valid := 1, [398].log_data[10].valid := 1, [398].log_data[11].valid := 1, [398].log_data[12].valid := 1, [398].log_data[13].valid := 1, [398].log_data[14].valid := 1, [398].log_data[15].valid := 1, [398].log_data[16].valid := 1, [398].log_data[17].valid := 1, [398].log_data[18].valid := 1, [398].log_data[19].valid := 1, [398].time.Year := 2023, [398].time.Month := 1, [398].time.Day := 19, [398].time.Hour := 9, [398].time.Minute := 34, [398].time.Second := 59, [399].log_data[0].min := 1.0, [399].log_data[0].max := 1.0, [399].log_data[0].total := 300.0, [399].log_data[0].time := 300.0, [399].log_data[0].minminute := 35, [399].log_data[0].maxminute := 35, [399].log_data[0].valid := 1, [399].log_data[1].valid := 1, [399].log_data[2].valid := 1, [399].log_data[3].valid := 1, [399].log_data[4].valid := 1, [399].log_data[5].valid := 1, [399].log_data[6].valid := 1, [399].log_data[7].valid := 1, [399].log_data[8].valid := 1, [399].log_data[9].valid := 1, [399].log_data[10].valid := 1, [399].log_data[11].valid := 1, [399].log_data[12].valid := 1, [399].log_data[13].valid := 1, [399].log_data[14].valid := 1, [399].log_data[15].valid := 1, [399].log_data[16].valid := 1, [399].log_data[17].valid := 1, [399].log_data[18].valid := 1, [399].log_data[19].valid := 1, [399].time.Year := 2023, [399].time.Month := 1, [399].time.Day := 19, [399].time.Hour := 9, [399].time.Minute := 39, [399].time.Second := 59, [400].log_data[0].min := 1.0, [400].log_data[0].max := 1.0, [400].log_data[0].total := 300.0, [400].log_data[0].time := 300.0, [400].log_data[0].minminute := 40, [400].log_data[0].maxminute := 40,
        [400].log_data[0].valid := 1, [400].log_data[1].valid := 1, [400].log_data[2].valid := 1, [400].log_data[3].valid := 1, [400].log_data[4].valid := 1, [400].log_data[5].valid := 1, [400].log_data[6].valid := 1, [400].log_data[7].valid := 1, [400].log_data[8].valid := 1, [400].log_data[9].valid := 1, [400].log_data[10].valid := 1, [400].log_data[11].valid := 1, [400].log_data[12].valid := 1, [400].log_data[13].valid := 1, [400].log_data[14].valid := 1, [400].log_data[15].valid := 1, [400].log_data[16].valid := 1, [400].log_data[17].valid := 1, [400].log_data[18].valid := 1, [400].log_data[19].valid := 1, [400].time.Year := 2023, [400].time.Month := 1, [400].time.Day := 19, [400].time.Hour := 9, [400].time.Minute := 44, [400].time.Second := 59, [401].log_data[0].min := 1.0, [401].log_data[0].max := 1.0, [401].log_data[0].total := 300.0, [401].log_data[0].time := 300.0, [401].log_data[0].minminute := 45, [401].log_data[0].maxminute := 45, [401].log_data[0].valid := 1, [401].log_data[1].valid := 1, [401].log_data[2].valid := 1, [401].log_data[3].valid := 1, [401].log_data[4].valid := 1, [401].log_data[5].valid := 1, [401].log_data[6].valid := 1, [401].log_data[7].valid := 1, [401].log_data[8].valid := 1, [401].log_data[9].valid := 1, [401].log_data[10].valid := 1, [401].log_data[11].valid := 1, [401].log_data[12].valid := 1, [401].log_data[13].valid := 1, [401].log_data[14].valid := 1, [401].log_data[15].valid := 1, [401].log_data[16].valid := 1, [401].log_data[17].valid := 1, [401].log_data[18].valid := 1, [401].log_data[19].valid := 1, [401].time.Year := 2023, [401].time.Month := 1, [401].time.Day := 19, [401].time.Hour := 9, [401].time.Minute := 49, [401].time.Second := 59, [402].log_data[0].min := 1.0, [402].log_data[0].max := 1.0,
        [402].log_data[0].total := 300.0, [402].log_data[0].time := 300.0, [402].log_data[0].minminute := 50, [402].log_data[0].maxminute := 50, [402].log_data[0].valid := 1, [402].log_data[1].valid := 1, [402].log_data[2].valid := 1, [402].log_data[3].valid := 1, [402].log_data[4].valid := 1, [402].log_data[5].valid := 1, [402].log_data[6].valid := 1, [402].log_data[7].valid := 1, [402].log_data[8].valid := 1, [402].log_data[9].valid := 1, [402].log_data[10].valid := 1, [402].log_data[11].valid := 1, [402].log_data[12].valid := 1, [402].log_data[13].valid := 1, [402].log_data[14].valid := 1, [402].log_data[15].valid := 1, [402].log_data[16].valid := 1, [402].log_data[17].valid := 1, [402].log_data[18].valid := 1, [402].log_data[19].valid := 1, [402].time.Year := 2023, [402].time.Month := 1, [402].time.Day := 19, [402].time.Hour := 9, [402].time.Minute := 54, [402].time.Second := 59, [403].log_data[0].min := 1.0, [403].log_data[0].max := 1.0, [403].log_data[0].total := 300.0, [403].log_data[0].time := 300.0, [403].log_data[0].minminute := 55, [403].log_data[0].maxminute := 55, [403].log_data[0].valid := 1, [403].log_data[1].valid := 1, [403].log_data[2].valid := 1, [403].log_data[3].valid := 1, [403].log_data[4].valid := 1, [403].log_data[5].valid := 1, [403].log_data[6].valid := 1, [403].log_data[7].valid := 1, [403].log_data[8].valid := 1, [403].log_data[9].valid := 1, [403].log_data[10].valid := 1, [403].log_data[11].valid := 1, [403].log_data[12].valid := 1, [403].log_data[13].valid := 1, [403].log_data[14].valid := 1, [403].log_data[15].valid := 1, [403].log_data[16].valid := 1, [403].log_data[17].valid := 1, [403].log_data[18].valid := 1, [403].log_data[19].valid := 1, [403].time.Year := 2023, [403].time.Month := 1, [403].time.Day := 19, [403].time.Hour := 9,
        [403].time.Minute := 59, [403].time.Second := 59, [404].log_data[0].min := 1.0, [404].log_data[0].max := 1.0, [404].log_data[0].total := 300.0, [404].log_data[0].time := 300.0, [404].log_data[0].valid := 1, [404].log_data[1].valid := 1, [404].log_data[2].valid := 1, [404].log_data[3].valid := 1, [404].log_data[4].valid := 1, [404].log_data[5].valid := 1, [404].log_data[6].valid := 1, [404].log_data[7].valid := 1, [404].log_data[8].valid := 1, [404].log_data[9].valid := 1, [404].log_data[10].valid := 1, [404].log_data[11].valid := 1, [404].log_data[12].valid := 1, [404].log_data[13].valid := 1, [404].log_data[14].valid := 1, [404].log_data[15].valid := 1, [404].log_data[16].valid := 1, [404].log_data[17].valid := 1, [404].log_data[18].valid := 1, [404].log_data[19].valid := 1, [404].time.Year := 2023, [404].time.Month := 1, [404].time.Day := 19, [404].time.Hour := 10, [404].time.Minute := 4, [404].time.Second := 59, [405].log_data[0].min := 1.0, [405].log_data[0].max := 1.0, [405].log_data[0].total := 300.0, [405].log_data[0].time := 300.0, [405].log_data[0].minminute := 5, [405].log_data[0].maxminute := 5, [405].log_data[0].valid := 1, [405].log_data[1].valid := 1, [405].log_data[2].valid := 1, [405].log_data[3].valid := 1, [405].log_data[4].valid := 1, [405].log_data[5].valid := 1, [405].log_data[6].valid := 1, [405].log_data[7].valid := 1, [405].log_data[8].valid := 1, [405].log_data[9].valid := 1, [405].log_data[10].valid := 1, [405].log_data[11].valid := 1, [405].log_data[12].valid := 1, [405].log_data[13].valid := 1, [405].log_data[14].valid := 1, [405].log_data[15].valid := 1, [405].log_data[16].valid := 1, [405].log_data[17].valid := 1, [405].log_data[18].valid := 1, [405].log_data[19].valid := 1, [405].time.Year := 2023, [405].time.Month := 1,
        [405].time.Day := 19, [405].time.Hour := 10, [405].time.Minute := 9, [405].time.Second := 59, [406].log_data[0].min := 1.0, [406].log_data[0].max := 1.0, [406].log_data[0].total := 300.0, [406].log_data[0].time := 300.0, [406].log_data[0].minminute := 10, [406].log_data[0].maxminute := 10, [406].log_data[0].valid := 1, [406].log_data[1].valid := 1, [406].log_data[2].valid := 1, [406].log_data[3].valid := 1, [406].log_data[4].valid := 1, [406].log_data[5].valid := 1, [406].log_data[6].valid := 1, [406].log_data[7].valid := 1, [406].log_data[8].valid := 1, [406].log_data[9].valid := 1, [406].log_data[10].valid := 1, [406].log_data[11].valid := 1, [406].log_data[12].valid := 1, [406].log_data[13].valid := 1, [406].log_data[14].valid := 1, [406].log_data[15].valid := 1, [406].log_data[16].valid := 1, [406].log_data[17].valid := 1, [406].log_data[18].valid := 1, [406].log_data[19].valid := 1, [406].time.Year := 2023, [406].time.Month := 1, [406].time.Day := 19, [406].time.Hour := 10, [406].time.Minute := 14, [406].time.Second := 59, [407].log_data[0].min := 1.0, [407].log_data[0].max := 1.0, [407].log_data[0].total := 300.0, [407].log_data[0].time := 300.0, [407].log_data[0].minminute := 15, [407].log_data[0].maxminute := 15, [407].log_data[0].valid := 1, [407].log_data[1].valid := 1, [407].log_data[2].valid := 1, [407].log_data[3].valid := 1, [407].log_data[4].valid := 1, [407].log_data[5].valid := 1, [407].log_data[6].valid := 1, [407].log_data[7].valid := 1, [407].log_data[8].valid := 1, [407].log_data[9].valid := 1, [407].log_data[10].valid := 1, [407].log_data[11].valid := 1, [407].log_data[12].valid := 1, [407].log_data[13].valid := 1, [407].log_data[14].valid := 1, [407].log_data[15].valid := 1, [407].log_data[16].valid := 1, [407].log_data[17].valid := 1,
        [407].log_data[18].valid := 1, [407].log_data[19].valid := 1, [407].time.Year := 2023, [407].time.Month := 1, [407].time.Day := 19, [407].time.Hour := 10, [407].time.Minute := 19, [407].time.Second := 59, [408].log_data[0].min := 1.0, [408].log_data[0].max := 1.0, [408].log_data[0].total := 300.0, [408].log_data[0].time := 300.0, [408].log_data[0].minminute := 20, [408].log_data[0].maxminute := 20, [408].log_data[0].valid := 1, [408].log_data[1].valid := 1, [408].log_data[2].valid := 1, [408].log_data[3].valid := 1, [408].log_data[4].valid := 1, [408].log_data[5].valid := 1, [408].log_data[6].valid := 1, [408].log_data[7].valid := 1, [408].log_data[8].valid := 1, [408].log_data[9].valid := 1, [408].log_data[10].valid := 1, [408].log_data[11].valid := 1, [408].log_data[12].valid := 1, [408].log_data[13].valid := 1, [408].log_data[14].valid := 1, [408].log_data[15].valid := 1, [408].log_data[16].valid := 1, [408].log_data[17].valid := 1, [408].log_data[18].valid := 1, [408].log_data[19].valid := 1, [408].time.Year := 2023, [408].time.Month := 1, [408].time.Day := 19, [408].time.Hour := 10, [408].time.Minute := 24, [408].time.Second := 59, [409].log_data[0].min := 1.0, [409].log_data[0].max := 1.0, [409].log_data[0].total := 300.0, [409].log_data[0].time := 300.0, [409].log_data[0].minminute := 25, [409].log_data[0].maxminute := 25, [409].log_data[0].valid := 1, [409].log_data[1].valid := 1, [409].log_data[2].valid := 1, [409].log_data[3].valid := 1, [409].log_data[4].valid := 1, [409].log_data[5].valid := 1, [409].log_data[6].valid := 1, [409].log_data[7].valid := 1, [409].log_data[8].valid := 1, [409].log_data[9].valid := 1, [409].log_data[10].valid := 1, [409].log_data[11].valid := 1, [409].log_data[12].valid := 1, [409].log_data[13].valid := 1,
        [409].log_data[14].valid := 1, [409].log_data[15].valid := 1, [409].log_data[16].valid := 1, [409].log_data[17].valid := 1, [409].log_data[18].valid := 1, [409].log_data[19].valid := 1, [409].time.Year := 2023, [409].time.Month := 1, [409].time.Day := 19, [409].time.Hour := 10, [409].time.Minute := 29, [409].time.Second := 59, [410].log_data[0].min := 1.0, [410].log_data[0].max := 1.0, [410].log_data[0].total := 300.0, [410].log_data[0].time := 300.0, [410].log_data[0].minminute := 30, [410].log_data[0].maxminute := 30, [410].log_data[0].valid := 1, [410].log_data[1].valid := 1, [410].log_data[2].valid := 1, [410].log_data[3].valid := 1, [410].log_data[4].valid := 1, [410].log_data[5].valid := 1, [410].log_data[6].valid := 1, [410].log_data[7].valid := 1, [410].log_data[8].valid := 1, [410].log_data[9].valid := 1, [410].log_data[10].valid := 1, [410].log_data[11].valid := 1, [410].log_data[12].valid := 1, [410].log_data[13].valid := 1, [410].log_data[14].valid := 1, [410].log_data[15].valid := 1, [410].log_data[16].valid := 1, [410].log_data[17].valid := 1, [410].log_data[18].valid := 1, [410].log_data[19].valid := 1, [410].time.Year := 2023, [410].time.Month := 1, [410].time.Day := 19, [410].time.Hour := 10, [410].time.Minute := 34, [410].time.Second := 59, [411].log_data[0].min := 1.0, [411].log_data[0].max := 1.0, [411].log_data[0].total := 300.0, [411].log_data[0].time := 300.0, [411].log_data[0].minminute := 35, [411].log_data[0].maxminute := 35, [411].log_data[0].valid := 1, [411].log_data[1].valid := 1, [411].log_data[2].valid := 1, [411].log_data[3].valid := 1, [411].log_data[4].valid := 1, [411].log_data[5].valid := 1, [411].log_data[6].valid := 1, [411].log_data[7].valid := 1, [411].log_data[8].valid := 1, [411].log_data[9].valid := 1,
        [411].log_data[10].valid := 1, [411].log_data[11].valid := 1, [411].log_data[12].valid := 1, [411].log_data[13].valid := 1, [411].log_data[14].valid := 1, [411].log_data[15].valid := 1, [411].log_data[16].valid := 1, [411].log_data[17].valid := 1, [411].log_data[18].valid := 1, [411].log_data[19].valid := 1, [411].time.Year := 2023, [411].time.Month := 1, [411].time.Day := 19, [411].time.Hour := 10, [411].time.Minute := 39, [411].time.Second := 59, [412].log_data[0].min := 1.0, [412].log_data[0].max := 1.0, [412].log_data[0].total := 300.0, [412].log_data[0].time := 300.0, [412].log_data[0].minminute := 40, [412].log_data[0].maxminute := 40, [412].log_data[0].valid := 1, [412].log_data[1].valid := 1, [412].log_data[2].valid := 1, [412].log_data[3].valid := 1, [412].log_data[4].valid := 1, [412].log_data[5].valid := 1, [412].log_data[6].valid := 1, [412].log_data[7].valid := 1, [412].log_data[8].valid := 1, [412].log_data[9].valid := 1, [412].log_data[10].valid := 1, [412].log_data[11].valid := 1, [412].log_data[12].valid := 1, [412].log_data[13].valid := 1, [412].log_data[14].valid := 1, [412].log_data[15].valid := 1, [412].log_data[16].valid := 1, [412].log_data[17].valid := 1, [412].log_data[18].valid := 1, [412].log_data[19].valid := 1, [412].time.Year := 2023, [412].time.Month := 1, [412].time.Day := 19, [412].time.Hour := 10, [412].time.Minute := 44, [412].time.Second := 59, [413].log_data[0].min := 1.0, [413].log_data[0].max := 1.0, [413].log_data[0].total := 300.0, [413].log_data[0].time := 300.0, [413].log_data[0].minminute := 45, [413].log_data[0].maxminute := 45, [413].log_data[0].valid := 1, [413].log_data[1].valid := 1, [413].log_data[2].valid := 1, [413].log_data[3].valid := 1, [413].log_data[4].valid := 1, [413].log_data[5].valid := 1,
        [413].log_data[6].valid := 1, [413].log_data[7].valid := 1, [413].log_data[8].valid := 1, [413].log_data[9].valid := 1, [413].log_data[10].valid := 1, [413].log_data[11].valid := 1, [413].log_data[12].valid := 1, [413].log_data[13].valid := 1, [413].log_data[14].valid := 1, [413].log_data[15].valid := 1, [413].log_data[16].valid := 1, [413].log_data[17].valid := 1, [413].log_data[18].valid := 1, [413].log_data[19].valid := 1, [413].time.Year := 2023, [413].time.Month := 1, [413].time.Day := 19, [413].time.Hour := 10, [413].time.Minute := 49, [413].time.Second := 59, [414].log_data[0].min := 1.0, [414].log_data[0].max := 1.0, [414].log_data[0].total := 300.0, [414].log_data[0].time := 300.0, [414].log_data[0].minminute := 50, [414].log_data[0].maxminute := 50, [414].log_data[0].valid := 1, [414].log_data[1].valid := 1, [414].log_data[2].valid := 1, [414].log_data[3].valid := 1, [414].log_data[4].valid := 1, [414].log_data[5].valid := 1, [414].log_data[6].valid := 1, [414].log_data[7].valid := 1, [414].log_data[8].valid := 1, [414].log_data[9].valid := 1, [414].log_data[10].valid := 1, [414].log_data[11].valid := 1, [414].log_data[12].valid := 1, [414].log_data[13].valid := 1, [414].log_data[14].valid := 1, [414].log_data[15].valid := 1, [414].log_data[16].valid := 1, [414].log_data[17].valid := 1, [414].log_data[18].valid := 1, [414].log_data[19].valid := 1, [414].time.Year := 2023, [414].time.Month := 1, [414].time.Day := 19, [414].time.Hour := 10, [414].time.Minute := 54, [414].time.Second := 59, [415].log_data[0].min := 1.0, [415].log_data[0].max := 1.0, [415].log_data[0].total := 300.0, [415].log_data[0].time := 300.0, [415].log_data[0].minminute := 55, [415].log_data[0].maxminute := 55, [415].log_data[0].valid := 1, [415].log_data[1].valid := 1,
        [415].log_data[2].valid := 1, [415].log_data[3].valid := 1, [415].log_data[4].valid := 1, [415].log_data[5].valid := 1, [415].log_data[6].valid := 1, [415].log_data[7].valid := 1, [415].log_data[8].valid := 1, [415].log_data[9].valid := 1, [415].log_data[10].valid := 1, [415].log_data[11].valid := 1, [415].log_data[12].valid := 1, [415].log_data[13].valid := 1, [415].log_data[14].valid := 1, [415].log_data[15].valid := 1, [415].log_data[16].valid := 1, [415].log_data[17].valid := 1, [415].log_data[18].valid := 1, [415].log_data[19].valid := 1, [415].time.Year := 2023, [415].time.Month := 1, [415].time.Day := 19, [415].time.Hour := 10, [415].time.Minute := 59, [415].time.Second := 59, [416].log_data[0].min := 1.0, [416].log_data[0].max := 1.0, [416].log_data[0].total := 300.0, [416].log_data[0].time := 300.0, [416].log_data[0].valid := 1, [416].log_data[1].valid := 1, [416].log_data[2].valid := 1, [416].log_data[3].valid := 1, [416].log_data[4].valid := 1, [416].log_data[5].valid := 1, [416].log_data[6].valid := 1, [416].log_data[7].valid := 1, [416].log_data[8].valid := 1, [416].log_data[9].valid := 1, [416].log_data[10].valid := 1, [416].log_data[11].valid := 1, [416].log_data[12].valid := 1, [416].log_data[13].valid := 1, [416].log_data[14].valid := 1, [416].log_data[15].valid := 1, [416].log_data[16].valid := 1, [416].log_data[17].valid := 1, [416].log_data[18].valid := 1, [416].log_data[19].valid := 1, [416].time.Year := 2023, [416].time.Month := 1, [416].time.Day := 19, [416].time.Hour := 11, [416].time.Minute := 4, [416].time.Second := 59, [417].log_data[0].min := 1.0, [417].log_data[0].max := 1.0, [417].log_data[0].total := 300.0, [417].log_data[0].time := 300.0, [417].log_data[0].minminute := 5, [417].log_data[0].maxminute := 5,
        [417].log_data[0].valid := 1, [417].log_data[1].valid := 1, [417].log_data[2].valid := 1, [417].log_data[3].valid := 1, [417].log_data[4].valid := 1, [417].log_data[5].valid := 1, [417].log_data[6].valid := 1, [417].log_data[7].valid := 1, [417].log_data[8].valid := 1, [417].log_data[9].valid := 1, [417].log_data[10].valid := 1, [417].log_data[11].valid := 1, [417].log_data[12].valid := 1, [417].log_data[13].valid := 1, [417].log_data[14].valid := 1, [417].log_data[15].valid := 1, [417].log_data[16].valid := 1, [417].log_data[17].valid := 1, [417].log_data[18].valid := 1, [417].log_data[19].valid := 1, [417].time.Year := 2023, [417].time.Month := 1, [417].time.Day := 19, [417].time.Hour := 11, [417].time.Minute := 9, [417].time.Second := 59, [418].log_data[0].min := 1.0, [418].log_data[0].max := 1.0, [418].log_data[0].total := 300.0, [418].log_data[0].time := 300.0, [418].log_data[0].minminute := 10, [418].log_data[0].maxminute := 10, [418].log_data[0].valid := 1, [418].log_data[1].valid := 1, [418].log_data[2].valid := 1, [418].log_data[3].valid := 1, [418].log_data[4].valid := 1, [418].log_data[5].valid := 1, [418].log_data[6].valid := 1, [418].log_data[7].valid := 1, [418].log_data[8].valid := 1, [418].log_data[9].valid := 1, [418].log_data[10].valid := 1, [418].log_data[11].valid := 1, [418].log_data[12].valid := 1, [418].log_data[13].valid := 1, [418].log_data[14].valid := 1, [418].log_data[15].valid := 1, [418].log_data[16].valid := 1, [418].log_data[17].valid := 1, [418].log_data[18].valid := 1, [418].log_data[19].valid := 1, [418].time.Year := 2023, [418].time.Month := 1, [418].time.Day := 19, [418].time.Hour := 11, [418].time.Minute := 14, [418].time.Second := 59, [419].log_data[0].min := 1.0, [419].log_data[0].max := 1.0,
        [419].log_data[0].total := 300.0, [419].log_data[0].time := 300.0, [419].log_data[0].minminute := 15, [419].log_data[0].maxminute := 15, [419].log_data[0].valid := 1, [419].log_data[1].valid := 1, [419].log_data[2].valid := 1, [419].log_data[3].valid := 1, [419].log_data[4].valid := 1, [419].log_data[5].valid := 1, [419].log_data[6].valid := 1, [419].log_data[7].valid := 1, [419].log_data[8].valid := 1, [419].log_data[9].valid := 1, [419].log_data[10].valid := 1, [419].log_data[11].valid := 1, [419].log_data[12].valid := 1, [419].log_data[13].valid := 1, [419].log_data[14].valid := 1, [419].log_data[15].valid := 1, [419].log_data[16].valid := 1, [419].log_data[17].valid := 1, [419].log_data[18].valid := 1, [419].log_data[19].valid := 1, [419].time.Year := 2023, [419].time.Month := 1, [419].time.Day := 19, [419].time.Hour := 11, [419].time.Minute := 19, [419].time.Second := 59, [420].log_data[0].min := 1.0, [420].log_data[0].max := 1.0, [420].log_data[0].total := 300.0, [420].log_data[0].time := 300.0, [420].log_data[0].minminute := 20, [420].log_data[0].maxminute := 20, [420].log_data[0].valid := 1, [420].log_data[1].valid := 1, [420].log_data[2].valid := 1, [420].log_data[3].valid := 1, [420].log_data[4].valid := 1, [420].log_data[5].valid := 1, [420].log_data[6].valid := 1, [420].log_data[7].valid := 1, [420].log_data[8].valid := 1, [420].log_data[9].valid := 1, [420].log_data[10].valid := 1, [420].log_data[11].valid := 1, [420].log_data[12].valid := 1, [420].log_data[13].valid := 1, [420].log_data[14].valid := 1, [420].log_data[15].valid := 1, [420].log_data[16].valid := 1, [420].log_data[17].valid := 1, [420].log_data[18].valid := 1, [420].log_data[19].valid := 1, [420].time.Year := 2023, [420].time.Month := 1, [420].time.Day := 19, [420].time.Hour := 11,
        [420].time.Minute := 24, [420].time.Second := 59, [421].log_data[0].min := 1.0, [421].log_data[0].max := 1.0, [421].log_data[0].total := 300.0, [421].log_data[0].time := 300.0, [421].log_data[0].minminute := 25, [421].log_data[0].maxminute := 25, [421].log_data[0].valid := 1, [421].log_data[1].valid := 1, [421].log_data[2].valid := 1, [421].log_data[3].valid := 1, [421].log_data[4].valid := 1, [421].log_data[5].valid := 1, [421].log_data[6].valid := 1, [421].log_data[7].valid := 1, [421].log_data[8].valid := 1, [421].log_data[9].valid := 1, [421].log_data[10].valid := 1, [421].log_data[11].valid := 1, [421].log_data[12].valid := 1, [421].log_data[13].valid := 1, [421].log_data[14].valid := 1, [421].log_data[15].valid := 1, [421].log_data[16].valid := 1, [421].log_data[17].valid := 1, [421].log_data[18].valid := 1, [421].log_data[19].valid := 1, [421].time.Year := 2023, [421].time.Month := 1, [421].time.Day := 19, [421].time.Hour := 11, [421].time.Minute := 29, [421].time.Second := 59, [422].log_data[0].min := 1.0, [422].log_data[0].max := 1.0, [422].log_data[0].total := 300.0, [422].log_data[0].time := 300.0, [422].log_data[0].minminute := 30, [422].log_data[0].maxminute := 30, [422].log_data[0].valid := 1, [422].log_data[1].valid := 1, [422].log_data[2].valid := 1, [422].log_data[3].valid := 1, [422].log_data[4].valid := 1, [422].log_data[5].valid := 1, [422].log_data[6].valid := 1, [422].log_data[7].valid := 1, [422].log_data[8].valid := 1, [422].log_data[9].valid := 1, [422].log_data[10].valid := 1, [422].log_data[11].valid := 1, [422].log_data[12].valid := 1, [422].log_data[13].valid := 1, [422].log_data[14].valid := 1, [422].log_data[15].valid := 1, [422].log_data[16].valid := 1, [422].log_data[17].valid := 1, [422].log_data[18].valid := 1, [422].log_data[19].valid := 1,
        [422].time.Year := 2023, [422].time.Month := 1, [422].time.Day := 19, [422].time.Hour := 11, [422].time.Minute := 34, [422].time.Second := 59, [423].log_data[0].min := 1.0, [423].log_data[0].max := 1.0, [423].log_data[0].total := 300.0, [423].log_data[0].time := 300.0, [423].log_data[0].minminute := 35, [423].log_data[0].maxminute := 35, [423].log_data[0].valid := 1, [423].log_data[1].valid := 1, [423].log_data[2].valid := 1, [423].log_data[3].valid := 1, [423].log_data[4].valid := 1, [423].log_data[5].valid := 1, [423].log_data[6].valid := 1, [423].log_data[7].valid := 1, [423].log_data[8].valid := 1, [423].log_data[9].valid := 1, [423].log_data[10].valid := 1, [423].log_data[11].valid := 1, [423].log_data[12].valid := 1, [423].log_data[13].valid := 1, [423].log_data[14].valid := 1, [423].log_data[15].valid := 1, [423].log_data[16].valid := 1, [423].log_data[17].valid := 1, [423].log_data[18].valid := 1, [423].log_data[19].valid := 1, [423].time.Year := 2023, [423].time.Month := 1, [423].time.Day := 19, [423].time.Hour := 11, [423].time.Minute := 39, [423].time.Second := 59, [424].log_data[0].min := 1.0, [424].log_data[0].max := 1.0, [424].log_data[0].total := 300.0, [424].log_data[0].time := 300.0, [424].log_data[0].minminute := 40, [424].log_data[0].maxminute := 40, [424].log_data[0].valid := 1, [424].log_data[1].valid := 1, [424].log_data[2].valid := 1, [424].log_data[3].valid := 1, [424].log_data[4].valid := 1, [424].log_data[5].valid := 1, [424].log_data[6].valid := 1, [424].log_data[7].valid := 1, [424].log_data[8].valid := 1, [424].log_data[9].valid := 1, [424].log_data[10].valid := 1, [424].log_data[11].valid := 1, [424].log_data[12].valid := 1, [424].log_data[13].valid := 1, [424].log_data[14].valid := 1, [424].log_data[15].valid := 1,
        [424].log_data[16].valid := 1, [424].log_data[17].valid := 1, [424].log_data[18].valid := 1, [424].log_data[19].valid := 1, [424].time.Year := 2023, [424].time.Month := 1, [424].time.Day := 19, [424].time.Hour := 11, [424].time.Minute := 44, [424].time.Second := 59, [425].log_data[0].min := 1.0, [425].log_data[0].max := 1.0, [425].log_data[0].total := 300.0, [425].log_data[0].time := 300.0, [425].log_data[0].minminute := 45, [425].log_data[0].maxminute := 45, [425].log_data[0].valid := 1, [425].log_data[1].valid := 1, [425].log_data[2].valid := 1, [425].log_data[3].valid := 1, [425].log_data[4].valid := 1, [425].log_data[5].valid := 1, [425].log_data[6].valid := 1, [425].log_data[7].valid := 1, [425].log_data[8].valid := 1, [425].log_data[9].valid := 1, [425].log_data[10].valid := 1, [425].log_data[11].valid := 1, [425].log_data[12].valid := 1, [425].log_data[13].valid := 1, [425].log_data[14].valid := 1, [425].log_data[15].valid := 1, [425].log_data[16].valid := 1, [425].log_data[17].valid := 1, [425].log_data[18].valid := 1, [425].log_data[19].valid := 1, [425].time.Year := 2023, [425].time.Month := 1, [425].time.Day := 19, [425].time.Hour := 11, [425].time.Minute := 49, [425].time.Second := 59, [426].log_data[0].min := 1.0, [426].log_data[0].max := 1.0, [426].log_data[0].total := 300.0, [426].log_data[0].time := 300.0, [426].log_data[0].minminute := 50, [426].log_data[0].maxminute := 50, [426].log_data[0].valid := 1, [426].log_data[1].valid := 1, [426].log_data[2].valid := 1, [426].log_data[3].valid := 1, [426].log_data[4].valid := 1, [426].log_data[5].valid := 1, [426].log_data[6].valid := 1, [426].log_data[7].valid := 1, [426].log_data[8].valid := 1, [426].log_data[9].valid := 1, [426].log_data[10].valid := 1, [426].log_data[11].valid := 1,
        [426].log_data[12].valid := 1, [426].log_data[13].valid := 1, [426].log_data[14].valid := 1, [426].log_data[15].valid := 1, [426].log_data[16].valid := 1, [426].log_data[17].valid := 1, [426].log_data[18].valid := 1, [426].log_data[19].valid := 1, [426].time.Year := 2023, [426].time.Month := 1, [426].time.Day := 19, [426].time.Hour := 11, [426].time.Minute := 54, [426].time.Second := 59, [427].log_data[0].min := 1.0, [427].log_data[0].max := 1.0, [427].log_data[0].total := 300.0, [427].log_data[0].time := 300.0, [427].log_data[0].minminute := 55, [427].log_data[0].maxminute := 55, [427].log_data[0].valid := 1, [427].log_data[1].valid := 1, [427].log_data[2].valid := 1, [427].log_data[3].valid := 1, [427].log_data[4].valid := 1, [427].log_data[5].valid := 1, [427].log_data[6].valid := 1, [427].log_data[7].valid := 1, [427].log_data[8].valid := 1, [427].log_data[9].valid := 1, [427].log_data[10].valid := 1, [427].log_data[11].valid := 1, [427].log_data[12].valid := 1, [427].log_data[13].valid := 1, [427].log_data[14].valid := 1, [427].log_data[15].valid := 1, [427].log_data[16].valid := 1, [427].log_data[17].valid := 1, [427].log_data[18].valid := 1, [427].log_data[19].valid := 1, [427].time.Year := 2023, [427].time.Month := 1, [427].time.Day := 19, [427].time.Hour := 11, [427].time.Minute := 59, [427].time.Second := 59, [428].log_data[0].min := 1.0, [428].log_data[0].max := 1.0, [428].log_data[0].total := 300.0, [428].log_data[0].time := 300.0, [428].log_data[0].valid := 1, [428].log_data[1].valid := 1, [428].log_data[2].valid := 1, [428].log_data[3].valid := 1, [428].log_data[4].valid := 1, [428].log_data[5].valid := 1, [428].log_data[6].valid := 1, [428].log_data[7].valid := 1, [428].log_data[8].valid := 1, [428].log_data[9].valid := 1,
        [428].log_data[10].valid := 1, [428].log_data[11].valid := 1, [428].log_data[12].valid := 1, [428].log_data[13].valid := 1, [428].log_data[14].valid := 1, [428].log_data[15].valid := 1, [428].log_data[16].valid := 1, [428].log_data[17].valid := 1, [428].log_data[18].valid := 1, [428].log_data[19].valid := 1, [428].time.Year := 2023, [428].time.Month := 1, [428].time.Day := 19, [428].time.Hour := 12, [428].time.Minute := 4, [428].time.Second := 59, [429].log_data[0].min := 1.0, [429].log_data[0].max := 1.0, [429].log_data[0].total := 300.0, [429].log_data[0].time := 300.0, [429].log_data[0].minminute := 5, [429].log_data[0].maxminute := 5, [429].log_data[0].valid := 1, [429].log_data[1].valid := 1, [429].log_data[2].valid := 1, [429].log_data[3].valid := 1, [429].log_data[4].valid := 1, [429].log_data[5].valid := 1, [429].log_data[6].valid := 1, [429].log_data[7].valid := 1, [429].log_data[8].valid := 1, [429].log_data[9].valid := 1, [429].log_data[10].valid := 1, [429].log_data[11].valid := 1, [429].log_data[12].valid := 1, [429].log_data[13].valid := 1, [429].log_data[14].valid := 1, [429].log_data[15].valid := 1, [429].log_data[16].valid := 1, [429].log_data[17].valid := 1, [429].log_data[18].valid := 1, [429].log_data[19].valid := 1, [429].time.Year := 2023, [429].time.Month := 1, [429].time.Day := 19, [429].time.Hour := 12, [429].time.Minute := 9, [429].time.Second := 59, [430].log_data[0].min := 1.0, [430].log_data[0].max := 1.0, [430].log_data[0].total := 300.0, [430].log_data[0].time := 300.0, [430].log_data[0].minminute := 10, [430].log_data[0].maxminute := 10, [430].log_data[0].valid := 1, [430].log_data[1].valid := 1, [430].log_data[2].valid := 1, [430].log_data[3].valid := 1, [430].log_data[4].valid := 1, [430].log_data[5].valid := 1,
        [430].log_data[6].valid := 1, [430].log_data[7].valid := 1, [430].log_data[8].valid := 1, [430].log_data[9].valid := 1, [430].log_data[10].valid := 1, [430].log_data[11].valid := 1, [430].log_data[12].valid := 1, [430].log_data[13].valid := 1, [430].log_data[14].valid := 1, [430].log_data[15].valid := 1, [430].log_data[16].valid := 1, [430].log_data[17].valid := 1, [430].log_data[18].valid := 1, [430].log_data[19].valid := 1, [430].time.Year := 2023, [430].time.Month := 1, [430].time.Day := 19, [430].time.Hour := 12, [430].time.Minute := 14, [430].time.Second := 59, [431].log_data[0].min := 1.0, [431].log_data[0].max := 1.0, [431].log_data[0].total := 300.0, [431].log_data[0].time := 300.0, [431].log_data[0].minminute := 15, [431].log_data[0].maxminute := 15, [431].log_data[0].valid := 1, [431].log_data[1].valid := 1, [431].log_data[2].valid := 1, [431].log_data[3].valid := 1, [431].log_data[4].valid := 1, [431].log_data[5].valid := 1, [431].log_data[6].valid := 1, [431].log_data[7].valid := 1, [431].log_data[8].valid := 1, [431].log_data[9].valid := 1, [431].log_data[10].valid := 1, [431].log_data[11].valid := 1, [431].log_data[12].valid := 1, [431].log_data[13].valid := 1, [431].log_data[14].valid := 1, [431].log_data[15].valid := 1, [431].log_data[16].valid := 1, [431].log_data[17].valid := 1, [431].log_data[18].valid := 1, [431].log_data[19].valid := 1, [431].time.Year := 2023, [431].time.Month := 1, [431].time.Day := 19, [431].time.Hour := 12, [431].time.Minute := 19, [431].time.Second := 59, [432].log_data[0].min := 1.0, [432].log_data[0].max := 1.0, [432].log_data[0].total := 300.0, [432].log_data[0].time := 300.0, [432].log_data[0].minminute := 20, [432].log_data[0].maxminute := 20, [432].log_data[0].valid := 1, [432].log_data[1].valid := 1,
        [432].log_data[2].valid := 1, [432].log_data[3].valid := 1, [432].log_data[4].valid := 1, [432].log_data[5].valid := 1, [432].log_data[6].valid := 1, [432].log_data[7].valid := 1, [432].log_data[8].valid := 1, [432].log_data[9].valid := 1, [432].log_data[10].valid := 1, [432].log_data[11].valid := 1, [432].log_data[12].valid := 1, [432].log_data[13].valid := 1, [432].log_data[14].valid := 1, [432].log_data[15].valid := 1, [432].log_data[16].valid := 1, [432].log_data[17].valid := 1, [432].log_data[18].valid := 1, [432].log_data[19].valid := 1, [432].time.Year := 2023, [432].time.Month := 1, [432].time.Day := 19, [432].time.Hour := 12, [432].time.Minute := 24, [432].time.Second := 59, [433].log_data[0].min := 1.0, [433].log_data[0].max := 1.0, [433].log_data[0].total := 300.0, [433].log_data[0].time := 300.0, [433].log_data[0].minminute := 25, [433].log_data[0].maxminute := 25, [433].log_data[0].valid := 1, [433].log_data[1].valid := 1, [433].log_data[2].valid := 1, [433].log_data[3].valid := 1, [433].log_data[4].valid := 1, [433].log_data[5].valid := 1, [433].log_data[6].valid := 1, [433].log_data[7].valid := 1, [433].log_data[8].valid := 1, [433].log_data[9].valid := 1, [433].log_data[10].valid := 1, [433].log_data[11].valid := 1, [433].log_data[12].valid := 1, [433].log_data[13].valid := 1, [433].log_data[14].valid := 1, [433].log_data[15].valid := 1, [433].log_data[16].valid := 1, [433].log_data[17].valid := 1, [433].log_data[18].valid := 1, [433].log_data[19].valid := 1, [433].time.Year := 2023, [433].time.Month := 1, [433].time.Day := 19, [433].time.Hour := 12, [433].time.Minute := 29, [433].time.Second := 59, [434].log_data[0].min := 1.0, [434].log_data[0].max := 1.0, [434].log_data[0].total := 300.0, [434].log_data[0].time := 300.0,
        [434].log_data[0].minminute := 30, [434].log_data[0].maxminute := 30, [434].log_data[0].valid := 1, [434].log_data[1].valid := 1, [434].log_data[2].valid := 1, [434].log_data[3].valid := 1, [434].log_data[4].valid := 1, [434].log_data[5].valid := 1, [434].log_data[6].valid := 1, [434].log_data[7].valid := 1, [434].log_data[8].valid := 1, [434].log_data[9].valid := 1, [434].log_data[10].valid := 1, [434].log_data[11].valid := 1, [434].log_data[12].valid := 1, [434].log_data[13].valid := 1, [434].log_data[14].valid := 1, [434].log_data[15].valid := 1, [434].log_data[16].valid := 1, [434].log_data[17].valid := 1, [434].log_data[18].valid := 1, [434].log_data[19].valid := 1, [434].time.Year := 2023, [434].time.Month := 1, [434].time.Day := 19, [434].time.Hour := 12, [434].time.Minute := 34, [434].time.Second := 59, [435].log_data[0].min := 1.0, [435].log_data[0].max := 1.0, [435].log_data[0].total := 300.0, [435].log_data[0].time := 300.0, [435].log_data[0].minminute := 35, [435].log_data[0].maxminute := 35, [435].log_data[0].valid := 1, [435].log_data[1].valid := 1, [435].log_data[2].valid := 1, [435].log_data[3].valid := 1, [435].log_data[4].valid := 1, [435].log_data[5].valid := 1, [435].log_data[6].valid := 1, [435].log_data[7].valid := 1, [435].log_data[8].valid := 1, [435].log_data[9].valid := 1, [435].log_data[10].valid := 1, [435].log_data[11].valid := 1, [435].log_data[12].valid := 1, [435].log_data[13].valid := 1, [435].log_data[14].valid := 1, [435].log_data[15].valid := 1, [435].log_data[16].valid := 1, [435].log_data[17].valid := 1, [435].log_data[18].valid := 1, [435].log_data[19].valid := 1, [435].time.Year := 2023, [435].time.Month := 1, [435].time.Day := 19, [435].time.Hour := 12, [435].time.Minute := 39, [435].time.Second := 59,
        [436].log_data[0].min := 1.0, [436].log_data[0].max := 1.0, [436].log_data[0].total := 300.0, [436].log_data[0].time := 300.0, [436].log_data[0].minminute := 40, [436].log_data[0].maxminute := 40, [436].log_data[0].valid := 1, [436].log_data[1].valid := 1, [436].log_data[2].valid := 1, [436].log_data[3].valid := 1, [436].log_data[4].valid := 1, [436].log_data[5].valid := 1, [436].log_data[6].valid := 1, [436].log_data[7].valid := 1, [436].log_data[8].valid := 1, [436].log_data[9].valid := 1, [436].log_data[10].valid := 1, [436].log_data[11].valid := 1, [436].log_data[12].valid := 1, [436].log_data[13].valid := 1, [436].log_data[14].valid := 1, [436].log_data[15].valid := 1, [436].log_data[16].valid := 1, [436].log_data[17].valid := 1, [436].log_data[18].valid := 1, [436].log_data[19].valid := 1, [436].time.Year := 2023, [436].time.Month := 1, [436].time.Day := 19, [436].time.Hour := 12, [436].time.Minute := 44, [436].time.Second := 59, [437].log_data[0].min := 1.0, [437].log_data[0].max := 1.0, [437].log_data[0].total := 300.0, [437].log_data[0].time := 300.0, [437].log_data[0].minminute := 45, [437].log_data[0].maxminute := 45, [437].log_data[0].valid := 1, [437].log_data[1].valid := 1, [437].log_data[2].valid := 1, [437].log_data[3].valid := 1, [437].log_data[4].valid := 1, [437].log_data[5].valid := 1, [437].log_data[6].valid := 1, [437].log_data[7].valid := 1, [437].log_data[8].valid := 1, [437].log_data[9].valid := 1, [437].log_data[10].valid := 1, [437].log_data[11].valid := 1, [437].log_data[12].valid := 1, [437].log_data[13].valid := 1, [437].log_data[14].valid := 1, [437].log_data[15].valid := 1, [437].log_data[16].valid := 1, [437].log_data[17].valid := 1, [437].log_data[18].valid := 1, [437].log_data[19].valid := 1, [437].time.Year := 2023, [437].time.Month := 1,
        [437].time.Day := 19, [437].time.Hour := 12, [437].time.Minute := 49, [437].time.Second := 59, [438].log_data[0].min := 1.0, [438].log_data[0].max := 1.0, [438].log_data[0].total := 300.0, [438].log_data[0].time := 300.0, [438].log_data[0].minminute := 50, [438].log_data[0].maxminute := 50, [438].log_data[0].valid := 1, [438].log_data[1].valid := 1, [438].log_data[2].valid := 1, [438].log_data[3].valid := 1, [438].log_data[4].valid := 1, [438].log_data[5].valid := 1, [438].log_data[6].valid := 1, [438].log_data[7].valid := 1, [438].log_data[8].valid := 1, [438].log_data[9].valid := 1, [438].log_data[10].valid := 1, [438].log_data[11].valid := 1, [438].log_data[12].valid := 1, [438].log_data[13].valid := 1, [438].log_data[14].valid := 1, [438].log_data[15].valid := 1, [438].log_data[16].valid := 1, [438].log_data[17].valid := 1, [438].log_data[18].valid := 1, [438].log_data[19].valid := 1, [438].time.Year := 2023, [438].time.Month := 1, [438].time.Day := 19, [438].time.Hour := 12, [438].time.Minute := 54, [438].time.Second := 59, [439].log_data[0].min := 1.0, [439].log_data[0].max := 1.0, [439].log_data[0].total := 300.0, [439].log_data[0].time := 300.0, [439].log_data[0].minminute := 55, [439].log_data[0].maxminute := 55, [439].log_data[0].valid := 1, [439].log_data[1].valid := 1, [439].log_data[2].valid := 1, [439].log_data[3].valid := 1, [439].log_data[4].valid := 1, [439].log_data[5].valid := 1, [439].log_data[6].valid := 1, [439].log_data[7].valid := 1, [439].log_data[8].valid := 1, [439].log_data[9].valid := 1, [439].log_data[10].valid := 1, [439].log_data[11].valid := 1, [439].log_data[12].valid := 1, [439].log_data[13].valid := 1, [439].log_data[14].valid := 1, [439].log_data[15].valid := 1, [439].log_data[16].valid := 1, [439].log_data[17].valid := 1,
        [439].log_data[18].valid := 1, [439].log_data[19].valid := 1, [439].time.Year := 2023, [439].time.Month := 1, [439].time.Day := 19, [439].time.Hour := 12, [439].time.Minute := 59, [439].time.Second := 59, [440].log_data[0].min := 1.0, [440].log_data[0].max := 1.0, [440].log_data[0].total := 300.0, [440].log_data[0].time := 300.0, [440].log_data[0].valid := 1, [440].log_data[1].valid := 1, [440].log_data[2].valid := 1, [440].log_data[3].valid := 1, [440].log_data[4].valid := 1, [440].log_data[5].valid := 1, [440].log_data[6].valid := 1, [440].log_data[7].valid := 1, [440].log_data[8].valid := 1, [440].log_data[9].valid := 1, [440].log_data[10].valid := 1, [440].log_data[11].valid := 1, [440].log_data[12].valid := 1, [440].log_data[13].valid := 1, [440].log_data[14].valid := 1, [440].log_data[15].valid := 1, [440].log_data[16].valid := 1, [440].log_data[17].valid := 1, [440].log_data[18].valid := 1, [440].log_data[19].valid := 1, [440].time.Year := 2023, [440].time.Month := 1, [440].time.Day := 19, [440].time.Hour := 13, [440].time.Minute := 4, [440].time.Second := 59, [441].log_data[0].min := 1.0, [441].log_data[0].max := 1.0, [441].log_data[0].total := 300.0, [441].log_data[0].time := 300.0, [441].log_data[0].minminute := 5, [441].log_data[0].maxminute := 5, [441].log_data[0].valid := 1, [441].log_data[1].valid := 1, [441].log_data[2].valid := 1, [441].log_data[3].valid := 1, [441].log_data[4].valid := 1, [441].log_data[5].valid := 1, [441].log_data[6].valid := 1, [441].log_data[7].valid := 1, [441].log_data[8].valid := 1, [441].log_data[9].valid := 1, [441].log_data[10].valid := 1, [441].log_data[11].valid := 1, [441].log_data[12].valid := 1, [441].log_data[13].valid := 1, [441].log_data[14].valid := 1, [441].log_data[15].valid := 1,
        [441].log_data[16].valid := 1, [441].log_data[17].valid := 1, [441].log_data[18].valid := 1, [441].log_data[19].valid := 1, [441].time.Year := 2023, [441].time.Month := 1, [441].time.Day := 19, [441].time.Hour := 13, [441].time.Minute := 9, [441].time.Second := 59, [442].log_data[0].min := 1.0, [442].log_data[0].max := 1.0, [442].log_data[0].total := 300.0, [442].log_data[0].time := 300.0, [442].log_data[0].minminute := 10, [442].log_data[0].maxminute := 10, [442].log_data[0].valid := 1, [442].log_data[1].valid := 1, [442].log_data[2].valid := 1, [442].log_data[3].valid := 1, [442].log_data[4].valid := 1, [442].log_data[5].valid := 1, [442].log_data[6].valid := 1, [442].log_data[7].valid := 1, [442].log_data[8].valid := 1, [442].log_data[9].valid := 1, [442].log_data[10].valid := 1, [442].log_data[11].valid := 1, [442].log_data[12].valid := 1, [442].log_data[13].valid := 1, [442].log_data[14].valid := 1, [442].log_data[15].valid := 1, [442].log_data[16].valid := 1, [442].log_data[17].valid := 1, [442].log_data[18].valid := 1, [442].log_data[19].valid := 1, [442].time.Year := 2023, [442].time.Month := 1, [442].time.Day := 19, [442].time.Hour := 13, [442].time.Minute := 14, [442].time.Second := 59, [443].log_data[0].min := 1.0, [443].log_data[0].max := 1.0, [443].log_data[0].total := 300.0, [443].log_data[0].time := 300.0, [443].log_data[0].minminute := 15, [443].log_data[0].maxminute := 15, [443].log_data[0].valid := 1, [443].log_data[1].valid := 1, [443].log_data[2].valid := 1, [443].log_data[3].valid := 1, [443].log_data[4].valid := 1, [443].log_data[5].valid := 1, [443].log_data[6].valid := 1, [443].log_data[7].valid := 1, [443].log_data[8].valid := 1, [443].log_data[9].valid := 1, [443].log_data[10].valid := 1, [443].log_data[11].valid := 1,
        [443].log_data[12].valid := 1, [443].log_data[13].valid := 1, [443].log_data[14].valid := 1, [443].log_data[15].valid := 1, [443].log_data[16].valid := 1, [443].log_data[17].valid := 1, [443].log_data[18].valid := 1, [443].log_data[19].valid := 1, [443].time.Year := 2023, [443].time.Month := 1, [443].time.Day := 19, [443].time.Hour := 13, [443].time.Minute := 19, [443].time.Second := 59, [444].log_data[0].min := 1.0, [444].log_data[0].max := 1.0, [444].log_data[0].total := 300.0, [444].log_data[0].time := 300.0, [444].log_data[0].minminute := 20, [444].log_data[0].maxminute := 20, [444].log_data[0].valid := 1, [444].log_data[1].valid := 1, [444].log_data[2].valid := 1, [444].log_data[3].valid := 1, [444].log_data[4].valid := 1, [444].log_data[5].valid := 1, [444].log_data[6].valid := 1, [444].log_data[7].valid := 1, [444].log_data[8].valid := 1, [444].log_data[9].valid := 1, [444].log_data[10].valid := 1, [444].log_data[11].valid := 1, [444].log_data[12].valid := 1, [444].log_data[13].valid := 1, [444].log_data[14].valid := 1, [444].log_data[15].valid := 1, [444].log_data[16].valid := 1, [444].log_data[17].valid := 1, [444].log_data[18].valid := 1, [444].log_data[19].valid := 1, [444].time.Year := 2023, [444].time.Month := 1, [444].time.Day := 19, [444].time.Hour := 13, [444].time.Minute := 24, [444].time.Second := 59, [445].log_data[0].min := 1.0, [445].log_data[0].max := 1.0, [445].log_data[0].total := 300.0, [445].log_data[0].time := 300.0, [445].log_data[0].minminute := 25, [445].log_data[0].maxminute := 25, [445].log_data[0].valid := 1, [445].log_data[1].valid := 1, [445].log_data[2].valid := 1, [445].log_data[3].valid := 1, [445].log_data[4].valid := 1, [445].log_data[5].valid := 1, [445].log_data[6].valid := 1, [445].log_data[7].valid := 1,
        [445].log_data[8].valid := 1, [445].log_data[9].valid := 1, [445].log_data[10].valid := 1, [445].log_data[11].valid := 1, [445].log_data[12].valid := 1, [445].log_data[13].valid := 1, [445].log_data[14].valid := 1, [445].log_data[15].valid := 1, [445].log_data[16].valid := 1, [445].log_data[17].valid := 1, [445].log_data[18].valid := 1, [445].log_data[19].valid := 1, [445].time.Year := 2023, [445].time.Month := 1, [445].time.Day := 19, [445].time.Hour := 13, [445].time.Minute := 29, [445].time.Second := 59, [446].log_data[0].min := 1.0, [446].log_data[0].max := 1.0, [446].log_data[0].total := 300.0, [446].log_data[0].time := 300.0, [446].log_data[0].minminute := 30, [446].log_data[0].maxminute := 30, [446].log_data[0].valid := 1, [446].log_data[1].valid := 1, [446].log_data[2].valid := 1, [446].log_data[3].valid := 1, [446].log_data[4].valid := 1, [446].log_data[5].valid := 1, [446].log_data[6].valid := 1, [446].log_data[7].valid := 1, [446].log_data[8].valid := 1, [446].log_data[9].valid := 1, [446].log_data[10].valid := 1, [446].log_data[11].valid := 1, [446].log_data[12].valid := 1, [446].log_data[13].valid := 1, [446].log_data[14].valid := 1, [446].log_data[15].valid := 1, [446].log_data[16].valid := 1, [446].log_data[17].valid := 1, [446].log_data[18].valid := 1, [446].log_data[19].valid := 1, [446].time.Year := 2023, [446].time.Month := 1, [446].time.Day := 19, [446].time.Hour := 13, [446].time.Minute := 34, [446].time.Second := 59, [447].log_data[0].min := 1.0, [447].log_data[0].max := 1.0, [447].log_data[0].total := 300.0, [447].log_data[0].time := 300.0, [447].log_data[0].minminute := 35, [447].log_data[0].maxminute := 35, [447].log_data[0].valid := 1, [447].log_data[1].valid := 1, [447].log_data[2].valid := 1, [447].log_data[3].valid := 1,
        [447].log_data[4].valid := 1, [447].log_data[5].valid := 1, [447].log_data[6].valid := 1, [447].log_data[7].valid := 1, [447].log_data[8].valid := 1, [447].log_data[9].valid := 1, [447].log_data[10].valid := 1, [447].log_data[11].valid := 1, [447].log_data[12].valid := 1, [447].log_data[13].valid := 1, [447].log_data[14].valid := 1, [447].log_data[15].valid := 1, [447].log_data[16].valid := 1, [447].log_data[17].valid := 1, [447].log_data[18].valid := 1, [447].log_data[19].valid := 1, [447].time.Year := 2023, [447].time.Month := 1, [447].time.Day := 19, [447].time.Hour := 13, [447].time.Minute := 39, [447].time.Second := 59, [448].log_data[0].min := 1.0, [448].log_data[0].max := 1.0, [448].log_data[0].total := 300.0, [448].log_data[0].time := 300.0, [448].log_data[0].minminute := 40, [448].log_data[0].maxminute := 40, [448].log_data[0].valid := 1, [448].log_data[1].valid := 1, [448].log_data[2].valid := 1, [448].log_data[3].valid := 1, [448].log_data[4].valid := 1, [448].log_data[5].valid := 1, [448].log_data[6].valid := 1, [448].log_data[7].valid := 1, [448].log_data[8].valid := 1, [448].log_data[9].valid := 1, [448].log_data[10].valid := 1, [448].log_data[11].valid := 1, [448].log_data[12].valid := 1, [448].log_data[13].valid := 1, [448].log_data[14].valid := 1, [448].log_data[15].valid := 1, [448].log_data[16].valid := 1, [448].log_data[17].valid := 1, [448].log_data[18].valid := 1, [448].log_data[19].valid := 1, [448].time.Year := 2023, [448].time.Month := 1, [448].time.Day := 19, [448].time.Hour := 13, [448].time.Minute := 44, [448].time.Second := 59, [449].log_data[0].min := 1.0, [449].log_data[0].max := 1.0, [449].log_data[0].total := 300.0, [449].log_data[0].time := 300.0, [449].log_data[0].minminute := 45, [449].log_data[0].maxminute := 45,
        [449].log_data[0].valid := 1, [449].log_data[1].valid := 1, [449].log_data[2].valid := 1, [449].log_data[3].valid := 1, [449].log_data[4].valid := 1, [449].log_data[5].valid := 1, [449].log_data[6].valid := 1, [449].log_data[7].valid := 1, [449].log_data[8].valid := 1, [449].log_data[9].valid := 1, [449].log_data[10].valid := 1, [449].log_data[11].valid := 1, [449].log_data[12].valid := 1, [449].log_data[13].valid := 1, [449].log_data[14].valid := 1, [449].log_data[15].valid := 1, [449].log_data[16].valid := 1, [449].log_data[17].valid := 1, [449].log_data[18].valid := 1, [449].log_data[19].valid := 1, [449].time.Year := 2023, [449].time.Month := 1, [449].time.Day := 19, [449].time.Hour := 13, [449].time.Minute := 49, [449].time.Second := 59, [450].log_data[0].min := 1.0, [450].log_data[0].max := 1.0, [450].log_data[0].total := 300.0, [450].log_data[0].time := 300.0, [450].log_data[0].minminute := 50, [450].log_data[0].maxminute := 50, [450].log_data[0].valid := 1, [450].log_data[1].valid := 1, [450].log_data[2].valid := 1, [450].log_data[3].valid := 1, [450].log_data[4].valid := 1, [450].log_data[5].valid := 1, [450].log_data[6].valid := 1, [450].log_data[7].valid := 1, [450].log_data[8].valid := 1, [450].log_data[9].valid := 1, [450].log_data[10].valid := 1, [450].log_data[11].valid := 1, [450].log_data[12].valid := 1, [450].log_data[13].valid := 1, [450].log_data[14].valid := 1, [450].log_data[15].valid := 1, [450].log_data[16].valid := 1, [450].log_data[17].valid := 1, [450].log_data[18].valid := 1, [450].log_data[19].valid := 1, [450].time.Year := 2023, [450].time.Month := 1, [450].time.Day := 19, [450].time.Hour := 13, [450].time.Minute := 54, [450].time.Second := 59, [451].log_data[0].min := 1.0, [451].log_data[0].max := 1.0,
        [451].log_data[0].total := 300.0, [451].log_data[0].time := 300.0, [451].log_data[0].minminute := 55, [451].log_data[0].maxminute := 55, [451].log_data[0].valid := 1, [451].log_data[1].valid := 1, [451].log_data[2].valid := 1, [451].log_data[3].valid := 1, [451].log_data[4].valid := 1, [451].log_data[5].valid := 1, [451].log_data[6].valid := 1, [451].log_data[7].valid := 1, [451].log_data[8].valid := 1, [451].log_data[9].valid := 1, [451].log_data[10].valid := 1, [451].log_data[11].valid := 1, [451].log_data[12].valid := 1, [451].log_data[13].valid := 1, [451].log_data[14].valid := 1, [451].log_data[15].valid := 1, [451].log_data[16].valid := 1, [451].log_data[17].valid := 1, [451].log_data[18].valid := 1, [451].log_data[19].valid := 1, [451].time.Year := 2023, [451].time.Month := 1, [451].time.Day := 19, [451].time.Hour := 13, [451].time.Minute := 59, [451].time.Second := 59, [452].log_data[0].min := 1.0, [452].log_data[0].max := 1.0, [452].log_data[0].total := 300.0, [452].log_data[0].time := 300.0, [452].log_data[0].valid := 1, [452].log_data[1].valid := 1, [452].log_data[2].valid := 1, [452].log_data[3].valid := 1, [452].log_data[4].valid := 1, [452].log_data[5].valid := 1, [452].log_data[6].valid := 1, [452].log_data[7].valid := 1, [452].log_data[8].valid := 1, [452].log_data[9].valid := 1, [452].log_data[10].valid := 1, [452].log_data[11].valid := 1, [452].log_data[12].valid := 1, [452].log_data[13].valid := 1, [452].log_data[14].valid := 1, [452].log_data[15].valid := 1, [452].log_data[16].valid := 1, [452].log_data[17].valid := 1, [452].log_data[18].valid := 1, [452].log_data[19].valid := 1, [452].time.Year := 2023, [452].time.Month := 1, [452].time.Day := 19, [452].time.Hour := 14, [452].time.Minute := 4, [452].time.Second := 59,
        [453].log_data[0].min := 1.0, [453].log_data[0].max := 1.0, [453].log_data[0].total := 300.0, [453].log_data[0].time := 300.0, [453].log_data[0].minminute := 5, [453].log_data[0].maxminute := 5, [453].log_data[0].valid := 1, [453].log_data[1].valid := 1, [453].log_data[2].valid := 1, [453].log_data[3].valid := 1, [453].log_data[4].valid := 1, [453].log_data[5].valid := 1, [453].log_data[6].valid := 1, [453].log_data[7].valid := 1, [453].log_data[8].valid := 1, [453].log_data[9].valid := 1, [453].log_data[10].valid := 1, [453].log_data[11].valid := 1, [453].log_data[12].valid := 1, [453].log_data[13].valid := 1, [453].log_data[14].valid := 1, [453].log_data[15].valid := 1, [453].log_data[16].valid := 1, [453].log_data[17].valid := 1, [453].log_data[18].valid := 1, [453].log_data[19].valid := 1, [453].time.Year := 2023, [453].time.Month := 1, [453].time.Day := 19, [453].time.Hour := 14, [453].time.Minute := 9, [453].time.Second := 59, [454].log_data[0].min := 1.0, [454].log_data[0].max := 1.0, [454].log_data[0].total := 300.0, [454].log_data[0].time := 300.0, [454].log_data[0].minminute := 10, [454].log_data[0].maxminute := 10, [454].log_data[0].valid := 1, [454].log_data[1].valid := 1, [454].log_data[2].valid := 1, [454].log_data[3].valid := 1, [454].log_data[4].valid := 1, [454].log_data[5].valid := 1, [454].log_data[6].valid := 1, [454].log_data[7].valid := 1, [454].log_data[8].valid := 1, [454].log_data[9].valid := 1, [454].log_data[10].valid := 1, [454].log_data[11].valid := 1, [454].log_data[12].valid := 1, [454].log_data[13].valid := 1, [454].log_data[14].valid := 1, [454].log_data[15].valid := 1, [454].log_data[16].valid := 1, [454].log_data[17].valid := 1, [454].log_data[18].valid := 1, [454].log_data[19].valid := 1, [454].time.Year := 2023, [454].time.Month := 1,
        [454].time.Day := 19, [454].time.Hour := 14, [454].time.Minute := 14, [454].time.Second := 59, [455].log_data[0].min := 1.0, [455].log_data[0].max := 1.0, [455].log_data[0].total := 300.0, [455].log_data[0].time := 300.0, [455].log_data[0].minminute := 15, [455].log_data[0].maxminute := 15, [455].log_data[0].valid := 1, [455].log_data[1].valid := 1, [455].log_data[2].valid := 1, [455].log_data[3].valid := 1, [455].log_data[4].valid := 1, [455].log_data[5].valid := 1, [455].log_data[6].valid := 1, [455].log_data[7].valid := 1, [455].log_data[8].valid := 1, [455].log_data[9].valid := 1, [455].log_data[10].valid := 1, [455].log_data[11].valid := 1, [455].log_data[12].valid := 1, [455].log_data[13].valid := 1, [455].log_data[14].valid := 1, [455].log_data[15].valid := 1, [455].log_data[16].valid := 1, [455].log_data[17].valid := 1, [455].log_data[18].valid := 1, [455].log_data[19].valid := 1, [455].time.Year := 2023, [455].time.Month := 1, [455].time.Day := 19, [455].time.Hour := 14, [455].time.Minute := 19, [455].time.Second := 59, [456].log_data[0].min := 1.0, [456].log_data[0].max := 1.0, [456].log_data[0].total := 300.0, [456].log_data[0].time := 300.0, [456].log_data[0].minminute := 20, [456].log_data[0].maxminute := 20, [456].log_data[0].valid := 1, [456].log_data[1].valid := 1, [456].log_data[2].valid := 1, [456].log_data[3].valid := 1, [456].log_data[4].valid := 1, [456].log_data[5].valid := 1, [456].log_data[6].valid := 1, [456].log_data[7].valid := 1, [456].log_data[8].valid := 1, [456].log_data[9].valid := 1, [456].log_data[10].valid := 1, [456].log_data[11].valid := 1, [456].log_data[12].valid := 1, [456].log_data[13].valid := 1, [456].log_data[14].valid := 1, [456].log_data[15].valid := 1, [456].log_data[16].valid := 1, [456].log_data[17].valid := 1,
        [456].log_data[18].valid := 1, [456].log_data[19].valid := 1, [456].time.Year := 2023, [456].time.Month := 1, [456].time.Day := 19, [456].time.Hour := 14, [456].time.Minute := 24, [456].time.Second := 59, [457].log_data[0].min := 1.0, [457].log_data[0].max := 1.0, [457].log_data[0].total := 300.0, [457].log_data[0].time := 300.0, [457].log_data[0].minminute := 25, [457].log_data[0].maxminute := 25, [457].log_data[0].valid := 1, [457].log_data[1].valid := 1, [457].log_data[2].valid := 1, [457].log_data[3].valid := 1, [457].log_data[4].valid := 1, [457].log_data[5].valid := 1, [457].log_data[6].valid := 1, [457].log_data[7].valid := 1, [457].log_data[8].valid := 1, [457].log_data[9].valid := 1, [457].log_data[10].valid := 1, [457].log_data[11].valid := 1, [457].log_data[12].valid := 1, [457].log_data[13].valid := 1, [457].log_data[14].valid := 1, [457].log_data[15].valid := 1, [457].log_data[16].valid := 1, [457].log_data[17].valid := 1, [457].log_data[18].valid := 1, [457].log_data[19].valid := 1, [457].time.Year := 2023, [457].time.Month := 1, [457].time.Day := 19, [457].time.Hour := 14, [457].time.Minute := 29, [457].time.Second := 59, [458].log_data[0].min := 1.0, [458].log_data[0].max := 1.0, [458].log_data[0].total := 300.0, [458].log_data[0].time := 300.0, [458].log_data[0].minminute := 30, [458].log_data[0].maxminute := 30, [458].log_data[0].valid := 1, [458].log_data[1].valid := 1, [458].log_data[2].valid := 1, [458].log_data[3].valid := 1, [458].log_data[4].valid := 1, [458].log_data[5].valid := 1, [458].log_data[6].valid := 1, [458].log_data[7].valid := 1, [458].log_data[8].valid := 1, [458].log_data[9].valid := 1, [458].log_data[10].valid := 1, [458].log_data[11].valid := 1, [458].log_data[12].valid := 1, [458].log_data[13].valid := 1,
        [458].log_data[14].valid := 1, [458].log_data[15].valid := 1, [458].log_data[16].valid := 1, [458].log_data[17].valid := 1, [458].log_data[18].valid := 1, [458].log_data[19].valid := 1, [458].time.Year := 2023, [458].time.Month := 1, [458].time.Day := 19, [458].time.Hour := 14, [458].time.Minute := 34, [458].time.Second := 59, [459].log_data[0].min := 1.0, [459].log_data[0].max := 1.0, [459].log_data[0].total := 300.0, [459].log_data[0].time := 300.0, [459].log_data[0].minminute := 35, [459].log_data[0].maxminute := 35, [459].log_data[0].valid := 1, [459].log_data[1].valid := 1, [459].log_data[2].valid := 1, [459].log_data[3].valid := 1, [459].log_data[4].valid := 1, [459].log_data[5].valid := 1, [459].log_data[6].valid := 1, [459].log_data[7].valid := 1, [459].log_data[8].valid := 1, [459].log_data[9].valid := 1, [459].log_data[10].valid := 1, [459].log_data[11].valid := 1, [459].log_data[12].valid := 1, [459].log_data[13].valid := 1, [459].log_data[14].valid := 1, [459].log_data[15].valid := 1, [459].log_data[16].valid := 1, [459].log_data[17].valid := 1, [459].log_data[18].valid := 1, [459].log_data[19].valid := 1, [459].time.Year := 2023, [459].time.Month := 1, [459].time.Day := 19, [459].time.Hour := 14, [459].time.Minute := 39, [459].time.Second := 59, [460].log_data[0].min := 1.0, [460].log_data[0].max := 1.0, [460].log_data[0].total := 300.0, [460].log_data[0].time := 300.0, [460].log_data[0].minminute := 40, [460].log_data[0].maxminute := 40, [460].log_data[0].valid := 1, [460].log_data[1].valid := 1, [460].log_data[2].valid := 1, [460].log_data[3].valid := 1, [460].log_data[4].valid := 1, [460].log_data[5].valid := 1, [460].log_data[6].valid := 1, [460].log_data[7].valid := 1, [460].log_data[8].valid := 1, [460].log_data[9].valid := 1,
        [460].log_data[10].valid := 1, [460].log_data[11].valid := 1, [460].log_data[12].valid := 1, [460].log_data[13].valid := 1, [460].log_data[14].valid := 1, [460].log_data[15].valid := 1, [460].log_data[16].valid := 1, [460].log_data[17].valid := 1, [460].log_data[18].valid := 1, [460].log_data[19].valid := 1, [460].time.Year := 2023, [460].time.Month := 1, [460].time.Day := 19, [460].time.Hour := 14, [460].time.Minute := 44, [460].time.Second := 59, [461].log_data[0].min := 1.0, [461].log_data[0].max := 1.0, [461].log_data[0].total := 300.0, [461].log_data[0].time := 300.0, [461].log_data[0].minminute := 45, [461].log_data[0].maxminute := 45, [461].log_data[0].valid := 1, [461].log_data[1].valid := 1, [461].log_data[2].valid := 1, [461].log_data[3].valid := 1, [461].log_data[4].valid := 1, [461].log_data[5].valid := 1, [461].log_data[6].valid := 1, [461].log_data[7].valid := 1, [461].log_data[8].valid := 1, [461].log_data[9].valid := 1, [461].log_data[10].valid := 1, [461].log_data[11].valid := 1, [461].log_data[12].valid := 1, [461].log_data[13].valid := 1, [461].log_data[14].valid := 1, [461].log_data[15].valid := 1, [461].log_data[16].valid := 1, [461].log_data[17].valid := 1, [461].log_data[18].valid := 1, [461].log_data[19].valid := 1, [461].time.Year := 2023, [461].time.Month := 1, [461].time.Day := 19, [461].time.Hour := 14, [461].time.Minute := 49, [461].time.Second := 59, [462].log_data[0].min := 1.0, [462].log_data[0].max := 1.0, [462].log_data[0].total := 300.0, [462].log_data[0].time := 300.0, [462].log_data[0].minminute := 50, [462].log_data[0].maxminute := 50, [462].log_data[0].valid := 1, [462].log_data[1].valid := 1, [462].log_data[2].valid := 1, [462].log_data[3].valid := 1, [462].log_data[4].valid := 1, [462].log_data[5].valid := 1,
        [462].log_data[6].valid := 1, [462].log_data[7].valid := 1, [462].log_data[8].valid := 1, [462].log_data[9].valid := 1, [462].log_data[10].valid := 1, [462].log_data[11].valid := 1, [462].log_data[12].valid := 1, [462].log_data[13].valid := 1, [462].log_data[14].valid := 1, [462].log_data[15].valid := 1, [462].log_data[16].valid := 1, [462].log_data[17].valid := 1, [462].log_data[18].valid := 1, [462].log_data[19].valid := 1, [462].time.Year := 2023, [462].time.Month := 1, [462].time.Day := 19, [462].time.Hour := 14, [462].time.Minute := 54, [462].time.Second := 59, [463].log_data[0].min := 1.0, [463].log_data[0].max := 1.0, [463].log_data[0].total := 300.0, [463].log_data[0].time := 300.0, [463].log_data[0].minminute := 55, [463].log_data[0].maxminute := 55, [463].log_data[0].valid := 1, [463].log_data[1].valid := 1, [463].log_data[2].valid := 1, [463].log_data[3].valid := 1, [463].log_data[4].valid := 1, [463].log_data[5].valid := 1, [463].log_data[6].valid := 1, [463].log_data[7].valid := 1, [463].log_data[8].valid := 1, [463].log_data[9].valid := 1, [463].log_data[10].valid := 1, [463].log_data[11].valid := 1, [463].log_data[12].valid := 1, [463].log_data[13].valid := 1, [463].log_data[14].valid := 1, [463].log_data[15].valid := 1, [463].log_data[16].valid := 1, [463].log_data[17].valid := 1, [463].log_data[18].valid := 1, [463].log_data[19].valid := 1, [463].time.Year := 2023, [463].time.Month := 1, [463].time.Day := 19, [463].time.Hour := 14, [463].time.Minute := 59, [463].time.Second := 59, [464].log_data[0].min := 1.0, [464].log_data[0].max := 1.0, [464].log_data[0].total := 300.0, [464].log_data[0].time := 300.0, [464].log_data[0].valid := 1, [464].log_data[1].valid := 1, [464].log_data[2].valid := 1, [464].log_data[3].valid := 1,
        [464].log_data[4].valid := 1, [464].log_data[5].valid := 1, [464].log_data[6].valid := 1, [464].log_data[7].valid := 1, [464].log_data[8].valid := 1, [464].log_data[9].valid := 1, [464].log_data[10].valid := 1, [464].log_data[11].valid := 1, [464].log_data[12].valid := 1, [464].log_data[13].valid := 1, [464].log_data[14].valid := 1, [464].log_data[15].valid := 1, [464].log_data[16].valid := 1, [464].log_data[17].valid := 1, [464].log_data[18].valid := 1, [464].log_data[19].valid := 1, [464].time.Year := 2023, [464].time.Month := 1, [464].time.Day := 19, [464].time.Hour := 15, [464].time.Minute := 4, [464].time.Second := 59, [465].log_data[0].min := 1.0, [465].log_data[0].max := 1.0, [465].log_data[0].total := 300.0, [465].log_data[0].time := 300.0, [465].log_data[0].minminute := 5, [465].log_data[0].maxminute := 5, [465].log_data[0].valid := 1, [465].log_data[1].valid := 1, [465].log_data[2].valid := 1, [465].log_data[3].valid := 1, [465].log_data[4].valid := 1, [465].log_data[5].valid := 1, [465].log_data[6].valid := 1, [465].log_data[7].valid := 1, [465].log_data[8].valid := 1, [465].log_data[9].valid := 1, [465].log_data[10].valid := 1, [465].log_data[11].valid := 1, [465].log_data[12].valid := 1, [465].log_data[13].valid := 1, [465].log_data[14].valid := 1, [465].log_data[15].valid := 1, [465].log_data[16].valid := 1, [465].log_data[17].valid := 1, [465].log_data[18].valid := 1, [465].log_data[19].valid := 1, [465].time.Year := 2023, [465].time.Month := 1, [465].time.Day := 19, [465].time.Hour := 15, [465].time.Minute := 9, [465].time.Second := 59, [466].log_data[0].min := 1.0, [466].log_data[0].max := 1.0, [466].log_data[0].total := 300.0, [466].log_data[0].time := 300.0, [466].log_data[0].minminute := 10, [466].log_data[0].maxminute := 10,
